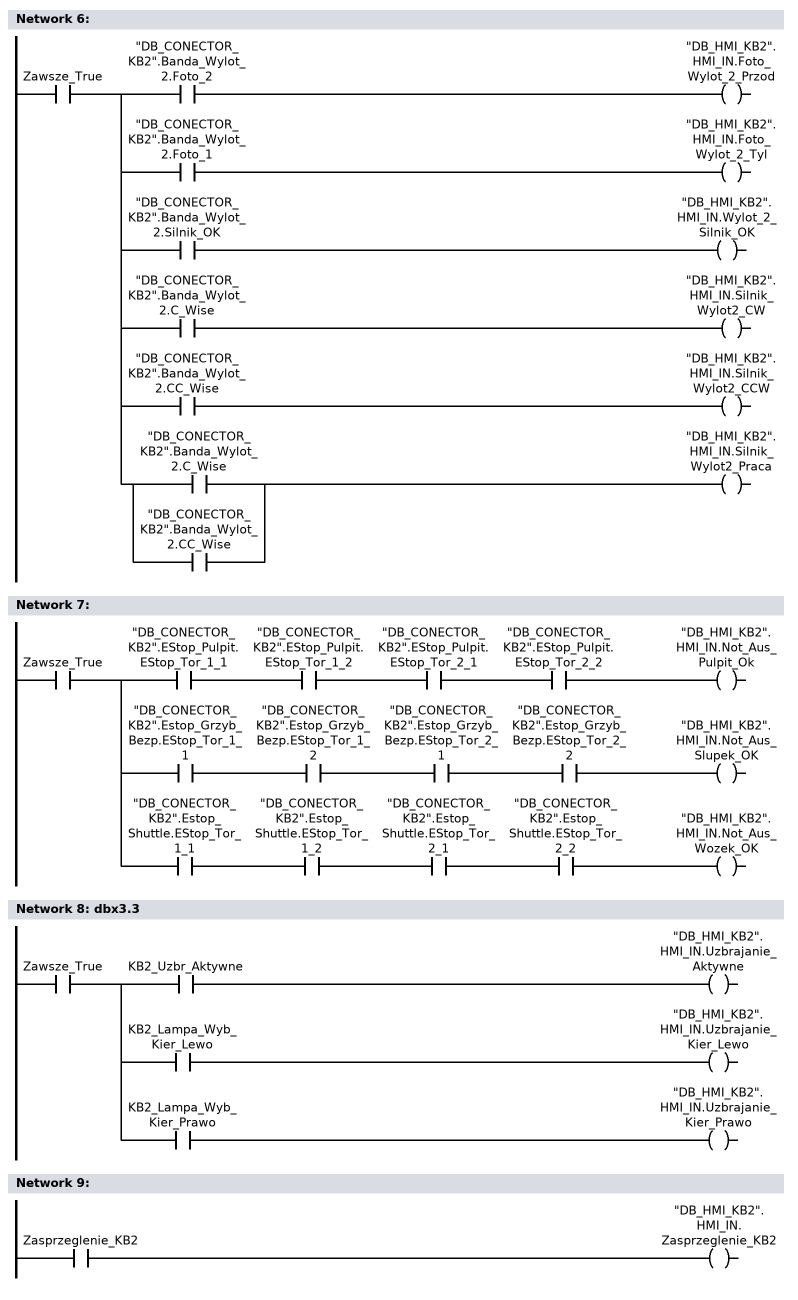
[picture p297: FC_HMI_KB2 networks 6-9]
NETWORK
TITLE =
//wylot 2
      A     "Zawsze_True";
      =     L 0.0;
      A     L 0.0;
      A     "DB_CONECTOR_KB2".Banda_Wylot_2.Foto_2;
      =     "DB_HMI_KB2".HMI_IN.Foto_Wylot_2_Przod;
      A     L 0.0;
      A     "DB_CONECTOR_KB2".Banda_Wylot_2.Foto_1;
      =     "DB_HMI_KB2".HMI_IN.Foto_Wylot_2_Tyl;
      A     L 0.0;
      A     "DB_CONECTOR_KB2".Banda_Wylot_2.Silnik_OK;
      =     "DB_HMI_KB2".HMI_IN.Wylot_2_Silnik_OK;
      A     L 0.0;
      A     "DB_CONECTOR_KB2".Banda_Wylot_2.C_Wise;
      =     "DB_HMI_KB2".HMI_IN.Silnik_Wylot2_CW;
      A     L 0.0;
      A     "DB_CONECTOR_KB2".Banda_Wylot_2.CC_Wise;
      =     "DB_HMI_KB2".HMI_IN.Silnik_Wylot2_CCW;
      A     L 0.0;
      A(;
      O     "DB_CONECTOR_KB2".Banda_Wylot_2.C_Wise;
      O     "DB_CONECTOR_KB2".Banda_Wylot_2.CC_Wise;
      );
      =     "DB_HMI_KB2".HMI_IN.Silnik_Wylot2_Praca;
NETWORK
TITLE =
//Not Aus pulpit
//
      A     "Zawsze_True";
      =     L 0.0;
      A     L 0.0;
      A     "DB_CONECTOR_KB2".EStop_Pulpit.EStop_Tor_1_1;
      A     "DB_CONECTOR_KB2".EStop_Pulpit.EStop_Tor_1_2;
      A     "DB_CONECTOR_KB2".EStop_Pulpit.EStop_Tor_2_1;
      A     "DB_CONECTOR_KB2".EStop_Pulpit.EStop_Tor_2_2;
      =     "DB_HMI_KB2".HMI_IN.Not_Aus_Pulpit_Ok;
      A     L 0.0;
      A     "DB_CONECTOR_KB2".Estop_Grzyb_Bezp.EStop_Tor_1_1;
      A     "DB_CONECTOR_KB2".Estop_Grzyb_Bezp.EStop_Tor_1_2;
      A     "DB_CONECTOR_KB2".Estop_Grzyb_Bezp.EStop_Tor_2_1;
      A     "DB_CONECTOR_KB2".Estop_Grzyb_Bezp.EStop_Tor_2_2;
      =     "DB_HMI_KB2".HMI_IN.Not_Aus_Slupek_OK;
      A     L 0.0;
      A     "DB_CONECTOR_KB2".Estop_Shuttle.EStop_Tor_1_1;
      A     "DB_CONECTOR_KB2".Estop_Shuttle.EStop_Tor_1_2;
      A     "DB_CONECTOR_KB2".Estop_Shuttle.EStop_Tor_2_1;
      A     "DB_CONECTOR_KB2".Estop_Shuttle.EStop_Tor_2_2;
      =     "DB_HMI_KB2".HMI_IN.Not_Aus_Wozek_OK;
NETWORK
TITLE = dbx3.3
//Uzbrajanie Aktywne
      A     "Zawsze_True";
      =     L 0.0;
      A     L 0.0;
      A     "KB2_Uzbr_Aktywne";
      =     "DB_HMI_KB2".HMI_IN.Uzbrajanie_Aktywne;
      A     L 0.0;
      A     "KB2_Lampa_Wyb_Kier_Lewo";
      =     "DB_HMI_KB2".HMI_IN.Uzbrajanie_Kier_Lewo;
      A     L 0.0;
      A     "KB2_Lampa_Wyb_Kier_Prawo";
      =     "DB_HMI_KB2".HMI_IN.Uzbrajanie_Kier_Prawo;
NETWORK
TITLE =
//Marka Zasprzeglenia KB2
      A     "Zasprzeglenie_KB2";
      =     "DB_HMI_KB2".HMI_IN.Zasprzeglenie_KB2;
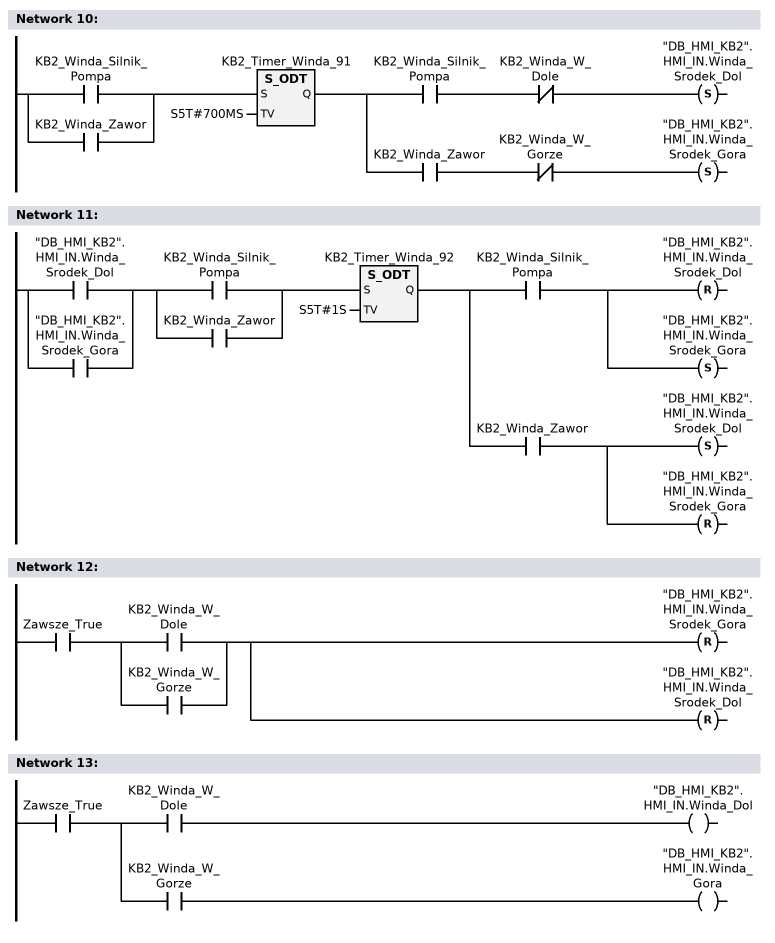
NETWORK
TITLE =
//Animacja windy
      A(;
      O     "KB2_Winda_Silnik_Pompa";
      O     "KB2_Winda_Zawor";
      );
      L     S5T#700MS;
      SD    "KB2_Timer_Winda_91";
      NOP   0;
      NOP   0;
      NOP   0;
      A     "KB2_Timer_Winda_91";
      =     L 0.0;
      A     L 0.0;
      A     "KB2_Winda_Silnik_Pompa";
      AN    "KB2_Winda_W_Dole";
      S     "DB_HMI_KB2".HMI_IN.Winda_Srodek_Dol;
      A     L 0.0;
      A     "KB2_Winda_Zawor";
      AN    "KB2_Winda_W_Gorze";
      S     "DB_HMI_KB2".HMI_IN.Winda_Srodek_Gora;
NETWORK
TITLE =
      A(;
      O     "DB_HMI_KB2".HMI_IN.Winda_Srodek_Dol;
      O     "DB_HMI_KB2".HMI_IN.Winda_Srodek_Gora;
      );
      A(;
      O     "KB2_Winda_Silnik_Pompa";
      O     "KB2_Winda_Zawor";
      );
      L     S5T#1S;
      SD    "KB2_Timer_Winda_92";
      NOP   0;
      NOP   0;
      NOP   0;
      A     "KB2_Timer_Winda_92";
      =     L 0.0;
      A     L 0.0;
      A     "KB2_Winda_Silnik_Pompa";
      R     "DB_HMI_KB2".HMI_IN.Winda_Srodek_Dol;
      S     "DB_HMI_KB2".HMI_IN.Winda_Srodek_Gora;
      A     L 0.0;
      A     "KB2_Winda_Zawor";
      S     "DB_HMI_KB2".HMI_IN.Winda_Srodek_Dol;
      R     "DB_HMI_KB2".HMI_IN.Winda_Srodek_Gora;
NETWORK
TITLE =
//Kasowanie skrajne winda
      A     "Zawsze_True";
      A(;
      O     "KB2_Winda_W_Dole";
      O     "KB2_Winda_W_Gorze";
      );
      R     "DB_HMI_KB2".HMI_IN.Winda_Srodek_Gora;
      R     "DB_HMI_KB2".HMI_IN.Winda_Srodek_Dol;
NETWORK
TITLE =
      A     "Zawsze_True";
      =     L 0.0;
      A     L 0.0;
      A     "KB2_Winda_W_Dole";
      =     "DB_HMI_KB2".HMI_IN.Winda_Dol;
      A     L 0.0;
      A     "KB2_Winda_W_Gorze";
      =     "DB_HMI_KB2".HMI_IN.Winda_Gora;
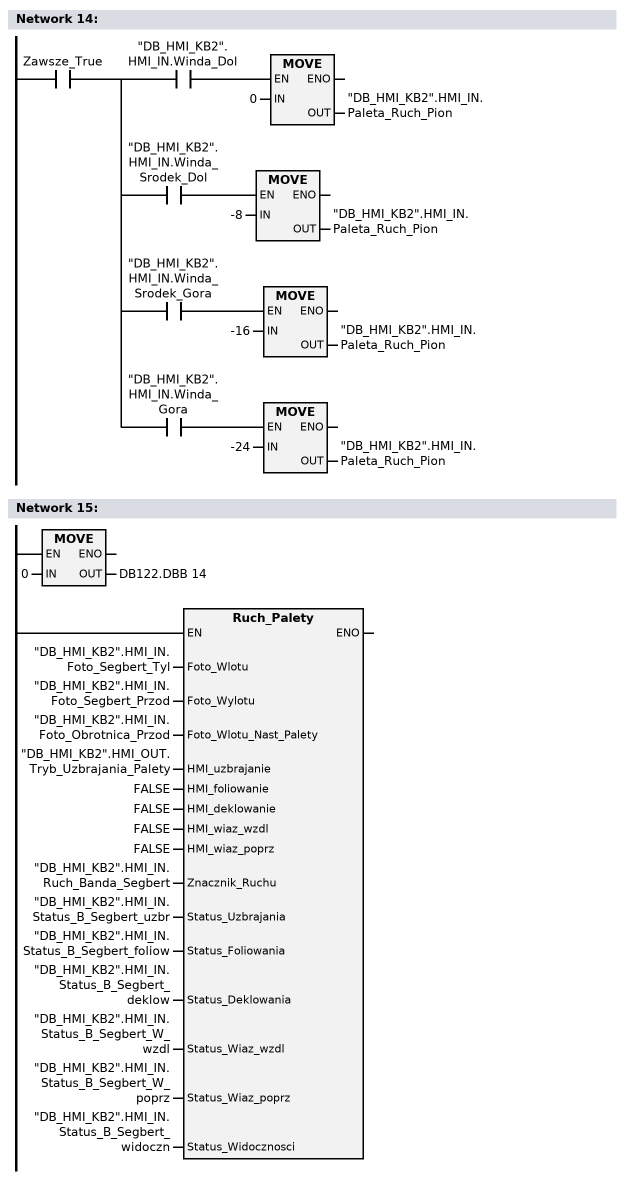
NETWORK
TITLE =
      A     "Zawsze_True";
      =     L 0.0;
      A     L 0.0;
      A     "DB_HMI_KB2".HMI_IN.Winda_Dol;
      JNB   _001;
      L     0;
      T     "DB_HMI_KB2".HMI_IN.Paleta_Ruch_Pion;
_001: NOP   0;
      A     L 0.0;
      A     "DB_HMI_KB2".HMI_IN.Winda_Srodek_Dol;
      JNB   _002;
      L     -8;
      T     "DB_HMI_KB2".HMI_IN.Paleta_Ruch_Pion;
_002: NOP   0;
      A     L 0.0;
      A     "DB_HMI_KB2".HMI_IN.Winda_Srodek_Gora;
      JNB   _003;
      L     -16;
      T     "DB_HMI_KB2".HMI_IN.Paleta_Ruch_Pion;
_003: NOP   0;
      A     L 0.0;
      A     "DB_HMI_KB2".HMI_IN.Winda_Gora;
      JNB   _004;
      L     -24;
      T     "DB_HMI_KB2".HMI_IN.Paleta_Ruch_Pion;
_004: NOP   0;
NETWORK
TITLE =
////Banda Segbert
      L     0;
      T     DB122.DBB 14;
      CALL  "Ruch_Palety" (
           Foto_Wlotu               := "DB_HMI_KB2".HMI_IN.Foto_Segbert_Tyl,
           Foto_Wylotu              := "DB_HMI_KB2".HMI_IN.Foto_Segbert_Przod,
           Foto_Wlotu_Nast_Palety   := "DB_HMI_KB2".HMI_IN.Foto_Obrotnica_Przod,
           HMI_uzbrajanie           := "DB_HMI_KB2".HMI_OUT.Tryb_Uzbrajania_Palety,
           HMI_foliowanie           := FALSE,
           HMI_deklowanie           := FALSE,
           HMI_wiaz_wzdl            := FALSE,
           HMI_wiaz_poprz           := FALSE,
           Znacznik_Ruchu           := "DB_HMI_KB2".HMI_IN.Ruch_Banda_Segbert,
           Status_Uzbrajania        := "DB_HMI_KB2".HMI_IN.Status_B_Segbert_uzbr,
           Status_Foliowania        := "DB_HMI_KB2".HMI_IN.Status_B_Segbert_foliow,
           Status_Deklowania        := "DB_HMI_KB2".HMI_IN.Status_B_Segbert_deklow,
           Status_Wiaz_wzdl         := "DB_HMI_KB2".HMI_IN.Status_B_Segbert_W_wzdl,
           Status_Wiaz_poprz        := "DB_HMI_KB2".HMI_IN.Status_B_Segbert_W_poprz,
           Status_Widocznosci       := "DB_HMI_KB2".HMI_IN.Status_B_Segbert_widoczn);
NETWORK
TITLE =
////Banda Obrotnica 0st
      L     0;
      T     DB122.DBB 15;
      A     DB122.DBX 7.0;
      JCN   et0;
      CALL  "Ruch_Palety" (
           Foto_Wlotu               := "DB_HMI_KB2".HMI_IN.Foto_Obrotnica_Przod,
           Foto_Wylotu              := "DB_HMI_KB2".HMI_IN.Foto_Obrotnica_Tyl,
           Foto_Wlotu_Nast_Palety   := "DB_HMI_KB2".HMI_IN.Foto_Winda_Tyl,
           HMI_uzbrajanie           := "DB_HMI_KB2".HMI_OUT.Tryb_Uzbrajania_Palety,
           HMI_foliowanie           := FALSE,
           HMI_deklowanie           := FALSE,
           HMI_wiaz_wzdl            := FALSE,
           HMI_wiaz_poprz           := FALSE,
           Znacznik_Ruchu           := "DB_HMI_KB2".HMI_IN.Ruch_Banda_Obrotnicy,
           Status_Uzbrajania        := "DB_HMI_KB2".HMI_IN.Status_B_Obr_0st_uzbr,
           Status_Foliowania        := "DB_HMI_KB2".HMI_IN.Status_B_Obr_0st_foliow,
           Status_Deklowania        := "DB_HMI_KB2".HMI_IN.Status_B_Obr_0st_deklow,
           Status_Wiaz_wzdl         := "DB_HMI_KB2".HMI_IN.Status_B_Obr_0st_W_wzdl,
           Status_Wiaz_poprz        := "DB_HMI_KB2".HMI_IN.Status_B_Obr_0st_W_poprz,
           Status_Widocznosci       := "DB_HMI_KB2".HMI_IN.Status_B_Obr_0st_widoczn);
      JU    ok0;
et0:  SET;
      R     "DB_HMI_KB2".HMI_IN.Status_B_Obr_0st_widoczn;
ok0:  NOP   0;
NETWORK
TITLE =
////Banda Obrotnica 90st
      L     0;
      T     DB122.DBB 19;
      A     DB122.DBX 8.0;
      JCN   et90;
      CALL  "Ruch_Palety" (
           Foto_Wlotu               := "DB_HMI_KB2".HMI_IN.Foto_Obrotnica_Przod,
           Foto_Wylotu              := "DB_HMI_KB2".HMI_IN.Foto_Obrotnica_Tyl,
           Foto_Wlotu_Nast_Palety   := "DB_HMI_KB2".HMI_IN.Foto_Wylot_2_Tyl,
           HMI_uzbrajanie           := "DB_HMI_KB2".HMI_OUT.Tryb_Uzbrajania_Palety,
           HMI_foliowanie           := FALSE,
           HMI_deklowanie           := FALSE,
           HMI_wiaz_wzdl            := FALSE,
           HMI_wiaz_poprz           := FALSE,
           Znacznik_Ruchu           := "DB_HMI_KB2".HMI_IN.Ruch_Banda_Obrotnicy,
           Status_Uzbrajania        := "DB_HMI_KB2".HMI_IN.Status_B_Obr_90st_uzbr,
           Status_Foliowania        := "DB_HMI_KB2".HMI_IN.Status_B_Obr_90st_foliow,
           Status_Deklowania        := "DB_HMI_KB2".HMI_IN.Status_B_Obr_90st_deklow,
           Status_Wiaz_wzdl         := "DB_HMI_KB2".HMI_IN.Status_B_Obr_90st_W_wzdl,
           Status_Wiaz_poprz        := "DB_HMI_KB2".HMI_IN.Status_B_Obr_90st_W_popr,
           Status_Widocznosci       := "DB_HMI_KB2".HMI_IN.Status_B_Obr_90st_widocz);
      JU    ok90;
et90: SET;
      R     "DB_HMI_KB2".HMI_IN.Status_B_Obr_90st_widocz;
ok90: NOP   0;
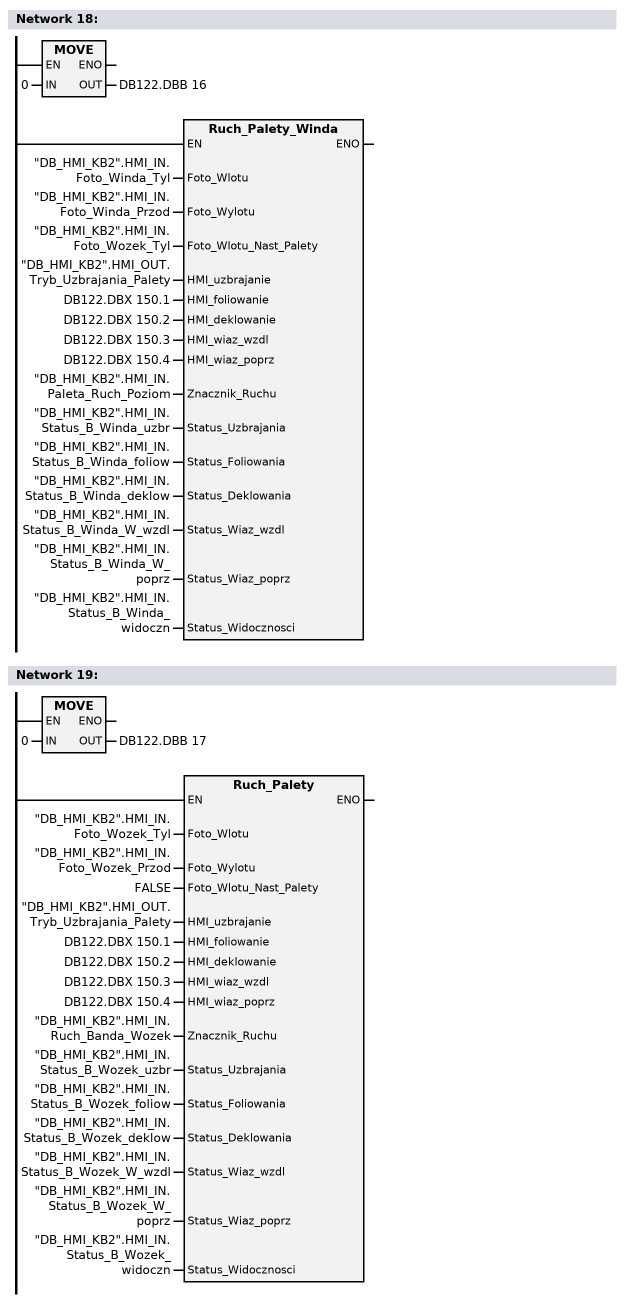
NETWORK
TITLE =
////Banda Winda
      L     0;
      T     DB122.DBB 16;
      CALL  "Ruch_Palety_Winda" (
           Foto_Wlotu               := "DB_HMI_KB2".HMI_IN.Foto_Winda_Tyl,
           Foto_Wylotu              := "DB_HMI_KB2".HMI_IN.Foto_Winda_Przod,
           Foto_Wlotu_Nast_Palety   := "DB_HMI_KB2".HMI_IN.Foto_Wozek_Tyl,
           HMI_uzbrajanie           := "DB_HMI_KB2".HMI_OUT.Tryb_Uzbrajania_Palety,
           HMI_foliowanie           := DB122.DBX 150.1,
           HMI_deklowanie           := DB122.DBX 150.2,
           HMI_wiaz_wzdl            := DB122.DBX 150.3,
           HMI_wiaz_poprz           := DB122.DBX 150.4,
           Znacznik_Ruchu           := "DB_HMI_KB2".HMI_IN.Paleta_Ruch_Poziom,
           Status_Uzbrajania        := "DB_HMI_KB2".HMI_IN.Status_B_Winda_uzbr,
           Status_Foliowania        := "DB_HMI_KB2".HMI_IN.Status_B_Winda_foliow,
           Status_Deklowania        := "DB_HMI_KB2".HMI_IN.Status_B_Winda_deklow,
           Status_Wiaz_wzdl         := "DB_HMI_KB2".HMI_IN.Status_B_Winda_W_wzdl,
           Status_Wiaz_poprz        := "DB_HMI_KB2".HMI_IN.Status_B_Winda_W_poprz,
           Status_Widocznosci       := "DB_HMI_KB2".HMI_IN.Status_B_Winda_widoczn);
NETWORK
TITLE =
////Banda Wozek
      L     0;
      T     DB122.DBB 17;
      CALL  "Ruch_Palety" (
           Foto_Wlotu               := "DB_HMI_KB2".HMI_IN.Foto_Wozek_Tyl,
           Foto_Wylotu              := "DB_HMI_KB2".HMI_IN.Foto_Wozek_Przod,
           Foto_Wlotu_Nast_Palety   := FALSE,
           HMI_uzbrajanie           := "DB_HMI_KB2".HMI_OUT.Tryb_Uzbrajania_Palety,
           HMI_foliowanie           := DB122.DBX 150.1,
           HMI_deklowanie           := DB122.DBX 150.2,
           HMI_wiaz_wzdl            := DB122.DBX 150.3,
           HMI_wiaz_poprz           := DB122.DBX 150.4,
           Znacznik_Ruchu           := "DB_HMI_KB2".HMI_IN.Ruch_Banda_Wozek,
           Status_Uzbrajania        := "DB_HMI_KB2".HMI_IN.Status_B_Wozek_uzbr,
           Status_Foliowania        := "DB_HMI_KB2".HMI_IN.Status_B_Wozek_foliow,
           Status_Deklowania        := "DB_HMI_KB2".HMI_IN.Status_B_Wozek_deklow,
           Status_Wiaz_wzdl         := "DB_HMI_KB2".HMI_IN.Status_B_Wozek_W_wzdl,
           Status_Wiaz_poprz        := "DB_HMI_KB2".HMI_IN.Status_B_Wozek_W_poprz,
           Status_Widocznosci       := "DB_HMI_KB2".HMI_IN.Status_B_Wozek_widoczn);
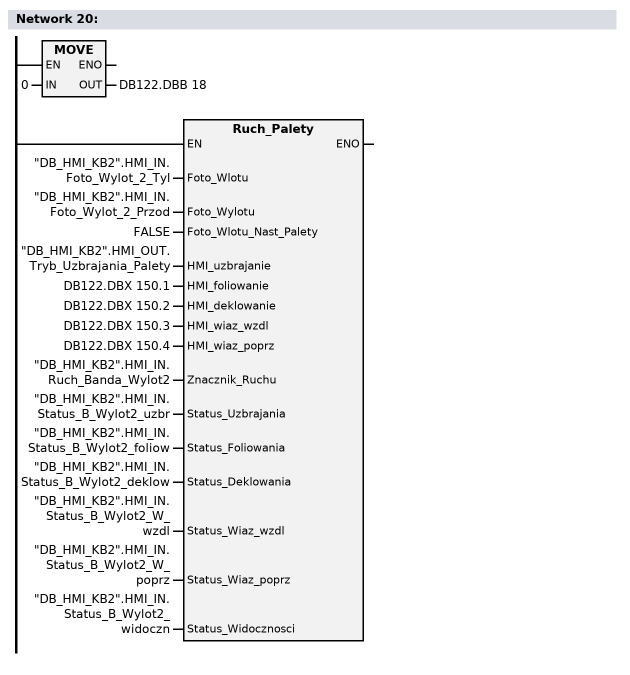
NETWORK
TITLE =
////Banda Wylot2
      L     0;
      T     DB122.DBB 18;
      CALL  "Ruch_Palety" (
           Foto_Wlotu               := "DB_HMI_KB2".HMI_IN.Foto_Wylot_2_Tyl,
           Foto_Wylotu              := "DB_HMI_KB2".HMI_IN.Foto_Wylot_2_Przod,
           Foto_Wlotu_Nast_Palety   := FALSE,
           HMI_uzbrajanie           := "DB_HMI_KB2".HMI_OUT.Tryb_Uzbrajania_Palety,
           HMI_foliowanie           := DB122.DBX 150.1,
           HMI_deklowanie           := DB122.DBX 150.2,
           HMI_wiaz_wzdl            := DB122.DBX 150.3,
           HMI_wiaz_poprz           := DB122.DBX 150.4,
           Znacznik_Ruchu           := "DB_HMI_KB2".HMI_IN.Ruch_Banda_Wylot2,
           Status_Uzbrajania        := "DB_HMI_KB2".HMI_IN.Status_B_Wylot2_uzbr,
           Status_Foliowania        := "DB_HMI_KB2".HMI_IN.Status_B_Wylot2_foliow,
           Status_Deklowania        := "DB_HMI_KB2".HMI_IN.Status_B_Wylot2_deklow,
           Status_Wiaz_wzdl         := "DB_HMI_KB2".HMI_IN.Status_B_Wylot2_W_wzdl,
           Status_Wiaz_poprz        := "DB_HMI_KB2".HMI_IN.Status_B_Wylot2_W_poprz,
           Status_Widocznosci       := "DB_HMI_KB2".HMI_IN.Status_B_Wylot2_widoczn);
END_FUNCTION

FUNCTION "FC_HMI_BUFF" : VOID	// FC 123
VERSION : 0.1
BEGIN
NETWORK
TITLE =
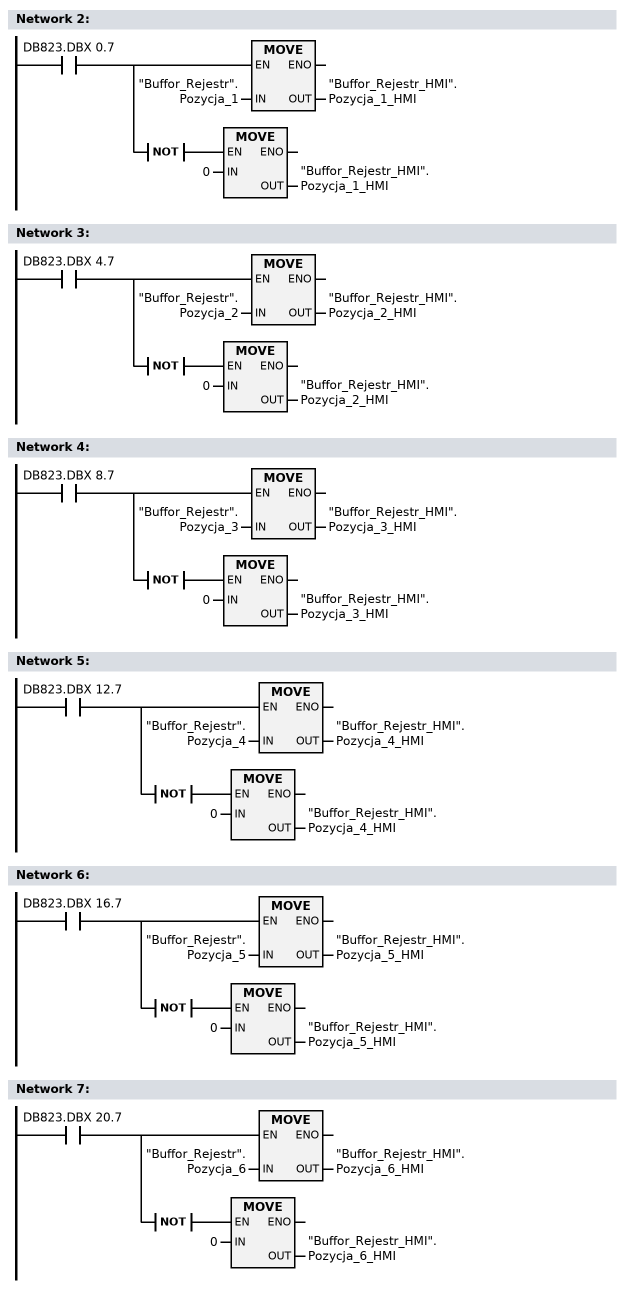
NETWORK
TITLE =
      A     DB823.DBX 0.7;
      =     L 0.0;
      A     L 0.0;
      JNB   _001;
      L     "Buffor_Rejestr".Pozycja_1;
      T     "Buffor_Rejestr_HMI".Pozycja_1_HMI;
_001: NOP   0;
      A     L 0.0;
      NOT;
      JNB   _008;
      L     0;
      T     "Buffor_Rejestr_HMI".Pozycja_1_HMI;
_008: NOP   0;
NETWORK
TITLE =
      A     DB823.DBX 4.7;
      =     L 0.0;
      A     L 0.0;
      JNB   _009;
      L     "Buffor_Rejestr".Pozycja_2;
      T     "Buffor_Rejestr_HMI".Pozycja_2_HMI;
_009: NOP   0;
      A     L 0.0;
      NOT;
      JNB   _00a;
      L     0;
      T     "Buffor_Rejestr_HMI".Pozycja_2_HMI;
_00a: NOP   0;
NETWORK
TITLE =
      A     DB823.DBX 8.7;
      =     L 0.0;
      A     L 0.0;
      JNB   _00b;
      L     "Buffor_Rejestr".Pozycja_3;
      T     "Buffor_Rejestr_HMI".Pozycja_3_HMI;
_00b: NOP   0;
      A     L 0.0;
      NOT;
      JNB   _00c;
      L     0;
      T     "Buffor_Rejestr_HMI".Pozycja_3_HMI;
_00c: NOP   0;
NETWORK
TITLE =
      A     DB823.DBX 12.7;
      =     L 0.0;
      A     L 0.0;
      JNB   _00d;
      L     "Buffor_Rejestr".Pozycja_4;
      T     "Buffor_Rejestr_HMI".Pozycja_4_HMI;
_00d: NOP   0;
      A     L 0.0;
      NOT;
      JNB   _00e;
      L     0;
      T     "Buffor_Rejestr_HMI".Pozycja_4_HMI;
_00e: NOP   0;
NETWORK
TITLE =
      A     DB823.DBX 16.7;
      =     L 0.0;
      A     L 0.0;
      JNB   _00f;
      L     "Buffor_Rejestr".Pozycja_5;
      T     "Buffor_Rejestr_HMI".Pozycja_5_HMI;
_00f: NOP   0;
      A     L 0.0;
      NOT;
      JNB   _010;
      L     0;
      T     "Buffor_Rejestr_HMI".Pozycja_5_HMI;
_010: NOP   0;
NETWORK
TITLE =
      A     DB823.DBX 20.7;
      =     L 0.0;
      A     L 0.0;
      JNB   _011;
      L     "Buffor_Rejestr".Pozycja_6;
      T     "Buffor_Rejestr_HMI".Pozycja_6_HMI;
_011: NOP   0;
      A     L 0.0;
      NOT;
      JNB   _012;
      L     0;
      T     "Buffor_Rejestr_HMI".Pozycja_6_HMI;
_012: NOP   0;
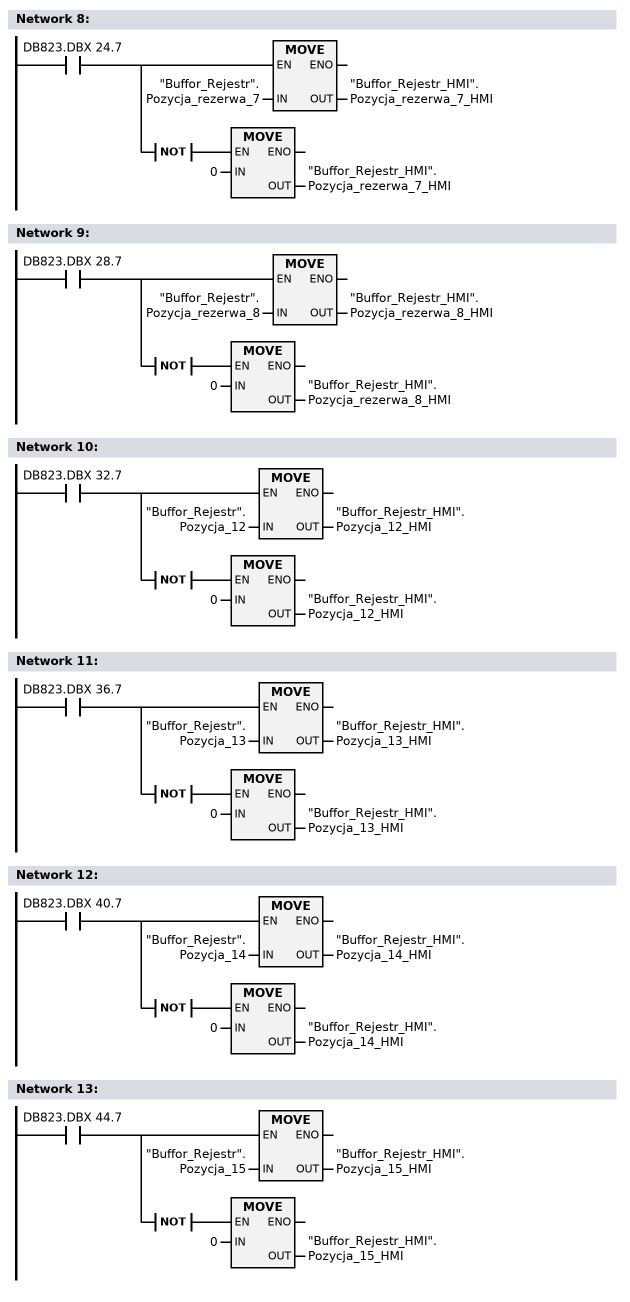
NETWORK
TITLE =
      A     DB823.DBX 24.7;
      =     L 0.0;
      A     L 0.0;
      JNB   _013;
      L     "Buffor_Rejestr".Pozycja_rezerwa_7;
      T     "Buffor_Rejestr_HMI".Pozycja_rezerwa_7_HMI;
_013: NOP   0;
      A     L 0.0;
      NOT;
      JNB   _014;
      L     0;
      T     "Buffor_Rejestr_HMI".Pozycja_rezerwa_7_HMI;
_014: NOP   0;
NETWORK
TITLE =
      A     DB823.DBX 28.7;
      =     L 0.0;
      A     L 0.0;
      JNB   _015;
      L     "Buffor_Rejestr".Pozycja_rezerwa_8;
      T     "Buffor_Rejestr_HMI".Pozycja_rezerwa_8_HMI;
_015: NOP   0;
      A     L 0.0;
      NOT;
      JNB   _016;
      L     0;
      T     "Buffor_Rejestr_HMI".Pozycja_rezerwa_8_HMI;
_016: NOP   0;
NETWORK
TITLE =
      A     DB823.DBX 32.7;
      =     L 0.0;
      A     L 0.0;
      JNB   _017;
      L     "Buffor_Rejestr".Pozycja_12;
      T     "Buffor_Rejestr_HMI".Pozycja_12_HMI;
_017: NOP   0;
      A     L 0.0;
      NOT;
      JNB   _018;
      L     0;
      T     "Buffor_Rejestr_HMI".Pozycja_12_HMI;
_018: NOP   0;
NETWORK
TITLE =
      A     DB823.DBX 36.7;
      =     L 0.0;
      A     L 0.0;
      JNB   _019;
      L     "Buffor_Rejestr".Pozycja_13;
      T     "Buffor_Rejestr_HMI".Pozycja_13_HMI;
_019: NOP   0;
      A     L 0.0;
      NOT;
      JNB   _01a;
      L     0;
      T     "Buffor_Rejestr_HMI".Pozycja_13_HMI;
_01a: NOP   0;
NETWORK
TITLE =
      A     DB823.DBX 40.7;
      =     L 0.0;
      A     L 0.0;
      JNB   _01b;
      L     "Buffor_Rejestr".Pozycja_14;
      T     "Buffor_Rejestr_HMI".Pozycja_14_HMI;
_01b: NOP   0;
      A     L 0.0;
      NOT;
      JNB   _01c;
      L     0;
      T     "Buffor_Rejestr_HMI".Pozycja_14_HMI;
_01c: NOP   0;
NETWORK
TITLE =
      A     DB823.DBX 44.7;
      =     L 0.0;
      A     L 0.0;
      JNB   _01d;
      L     "Buffor_Rejestr".Pozycja_15;
      T     "Buffor_Rejestr_HMI".Pozycja_15_HMI;
_01d: NOP   0;
      A     L 0.0;
      NOT;
      JNB   _01e;
      L     0;
      T     "Buffor_Rejestr_HMI".Pozycja_15_HMI;
_01e: NOP   0;
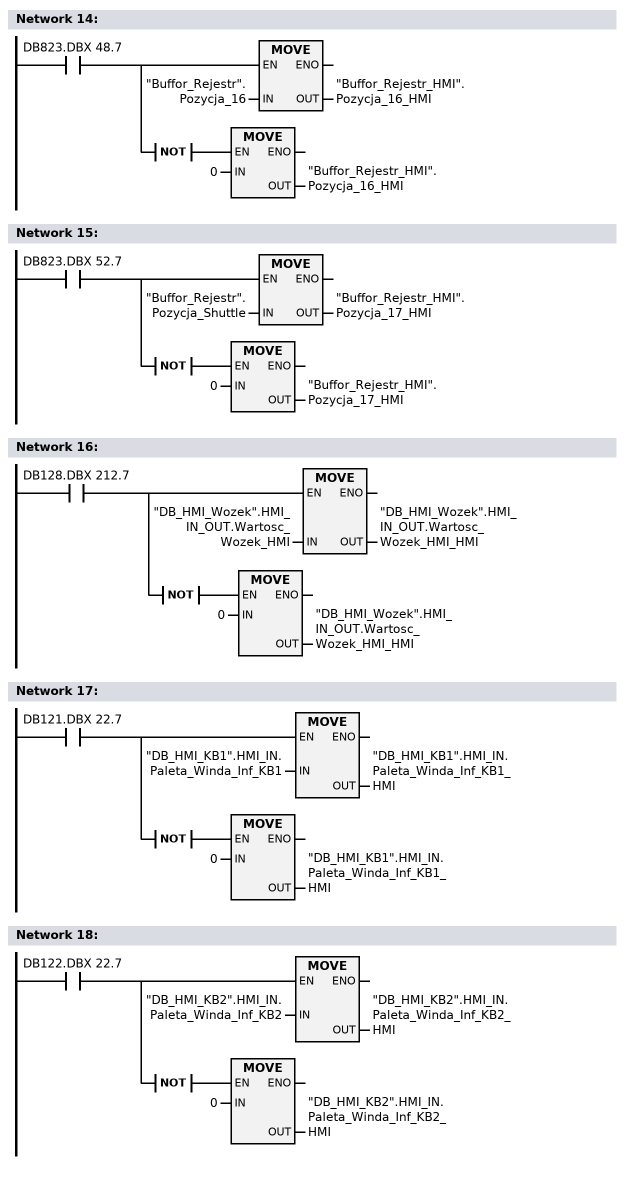
NETWORK
TITLE =
      A     DB823.DBX 48.7;
      =     L 0.0;
      A     L 0.0;
      JNB   _01f;
      L     "Buffor_Rejestr".Pozycja_16;
      T     "Buffor_Rejestr_HMI".Pozycja_16_HMI;
_01f: NOP   0;
      A     L 0.0;
      NOT;
      JNB   _020;
      L     0;
      T     "Buffor_Rejestr_HMI".Pozycja_16_HMI;
_020: NOP   0;
NETWORK
TITLE =
      A     DB823.DBX 52.7;
      =     L 0.0;
      A     L 0.0;
      JNB   _021;
      L     "Buffor_Rejestr".Pozycja_Shuttle;
      T     "Buffor_Rejestr_HMI".Pozycja_17_HMI;
_021: NOP   0;
      A     L 0.0;
      NOT;
      JNB   _022;
      L     0;
      T     "Buffor_Rejestr_HMI".Pozycja_17_HMI;
_022: NOP   0;
NETWORK
TITLE =
      A     DB128.DBX 212.7;
      =     L 0.0;
      A     L 0.0;
      JNB   _023;
      L     "DB_HMI_Wozek".HMI_IN_OUT.Wartosc_Wozek_HMI;
      T     "DB_HMI_Wozek".HMI_IN_OUT.Wartosc_Wozek_HMI_HMI;
_023: NOP   0;
      A     L 0.0;
      NOT;
      JNB   _024;
      L     0;
      T     "DB_HMI_Wozek".HMI_IN_OUT.Wartosc_Wozek_HMI_HMI;
_024: NOP   0;
NETWORK
TITLE =
      A     DB121.DBX 22.7;
      =     L 0.0;
      A     L 0.0;
      JNB   _025;
      L     "DB_HMI_KB1".HMI_IN.Paleta_Winda_Inf_KB1;
      T     "DB_HMI_KB1".HMI_IN.Paleta_Winda_Inf_KB1_HMI;
_025: NOP   0;
      A     L 0.0;
      NOT;
      JNB   _026;
      L     0;
      T     "DB_HMI_KB1".HMI_IN.Paleta_Winda_Inf_KB1_HMI;
_026: NOP   0;
NETWORK
TITLE =
      A     DB122.DBX 22.7;
      =     L 0.0;
      A     L 0.0;
      JNB   _027;
      L     "DB_HMI_KB2".HMI_IN.Paleta_Winda_Inf_KB2;
      T     "DB_HMI_KB2".HMI_IN.Paleta_Winda_Inf_KB2_HMI;
_027: NOP   0;
      A     L 0.0;
      NOT;
      JNB   _028;
      L     0;
      T     "DB_HMI_KB2".HMI_IN.Paleta_Winda_Inf_KB2_HMI;
_028: NOP   0;
END_FUNCTION

FUNCTION "FC_HMI_WOZEK" : VOID	// FC 128
AUTHOR : Kng
NAME : Main
VERSION : 0.1
VAR_TEMP
  Temp_Help_1 : BOOL ;
END_VAR
BEGIN
NETWORK
TITLE =
//Ten Network celowo jest wolny
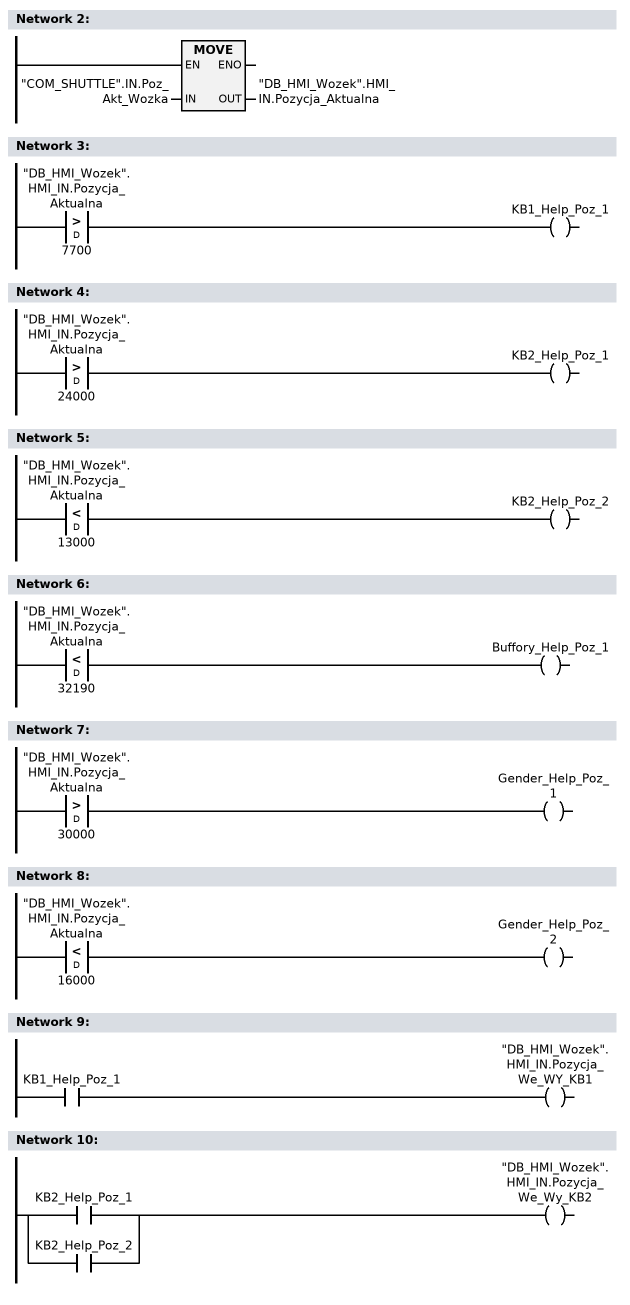
NETWORK
TITLE =
//Pozycja Aktualna
      L     "COM_SHUTTLE".IN.Poz_Akt_Wozka;
      T     "DB_HMI_Wozek".HMI_IN.Pozycja_Aktualna;
      NOP   0;
NETWORK
TITLE =
//wyznaczenie zakresu widzialnosci wozka na HMI dla KB1
      L     "DB_HMI_Wozek".HMI_IN.Pozycja_Aktualna;
      L     7700;
      >D;
      =     "KB1_Help_Poz_1";
NETWORK
TITLE =
//wyznaczenie zakresu widzialnosci wozka na HMI dla KB2
      L     "DB_HMI_Wozek".HMI_IN.Pozycja_Aktualna;
      L     24000;
      >D;
      =     "KB2_Help_Poz_1";
NETWORK
TITLE =
//wyznaczenie zakresu widzialnosci wozka na HMI dla KB2
      L     "DB_HMI_Wozek".HMI_IN.Pozycja_Aktualna;
      L     13000;
      <D;
      =     "KB2_Help_Poz_2";
NETWORK
TITLE =
//wyznaczenie zakresu widzialnosci wozka na HMI dla Buffory_Manual
//
      L     "DB_HMI_Wozek".HMI_IN.Pozycja_Aktualna;
      L     32190;
      <D;
      =     "Buffory_Help_Poz_1";
NETWORK
TITLE =
//wyznaczenie zakresu widzialnosci wozka na HMI dla Gender
      L     "DB_HMI_Wozek".HMI_IN.Pozycja_Aktualna;
      L     30000;
      >D;
      =     "Gender_Help_Poz_1";
NETWORK
TITLE =
//wyznaczenie zakresu widzialnosci wozka na HMI dla Gender
      L     "DB_HMI_Wozek".HMI_IN.Pozycja_Aktualna;
      L     16000;
      <D;
      =     "Gender_Help_Poz_2";
NETWORK
TITLE =
//wyznaczenie zakresu widzialnosci wozka na HMI dla KB1
      A     "KB1_Help_Poz_1";
      =     "DB_HMI_Wozek".HMI_IN.Pozycja_We_WY_KB1;
NETWORK
TITLE =
//wyznaczenie zakresu widzialnosci wozka na HMI dla KB2
      O     "KB2_Help_Poz_1";
      O     "KB2_Help_Poz_2";
      =     "DB_HMI_Wozek".HMI_IN.Pozycja_We_Wy_KB2;
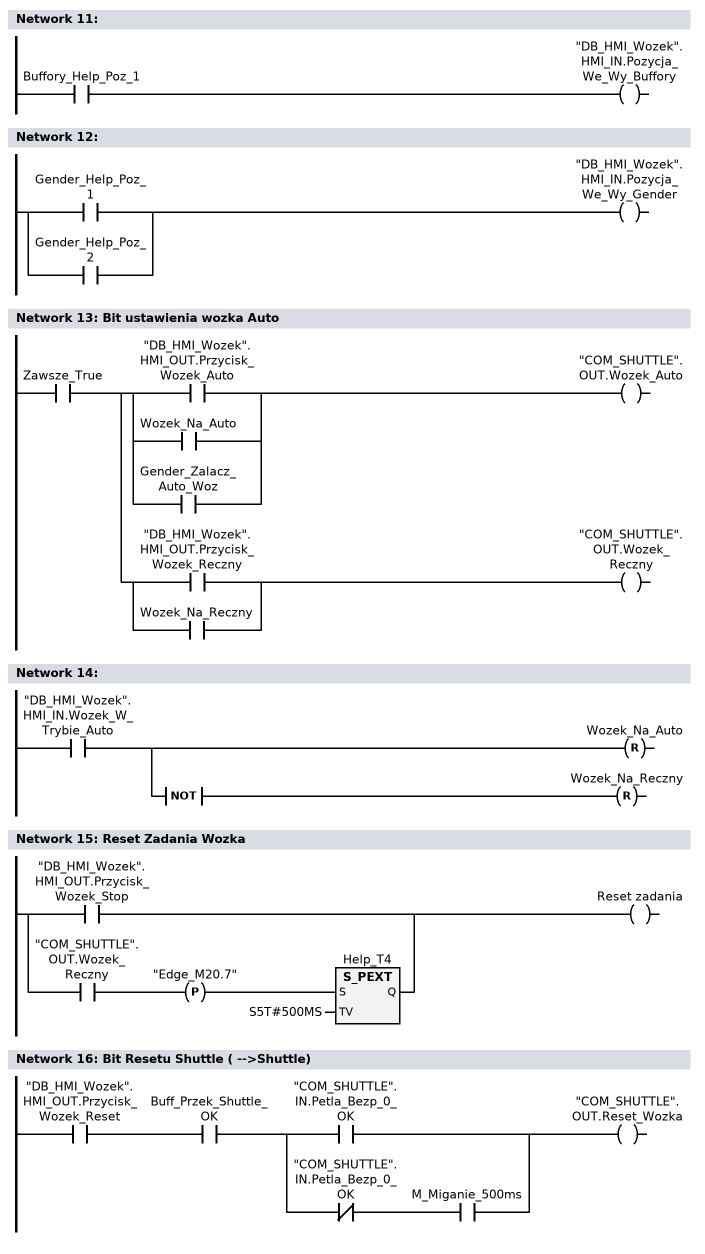
NETWORK
TITLE =
//wyznaczenie zakresu widzialnosci wozka na HMI dla Buffory_Manual
      A     "Buffory_Help_Poz_1";
      =     "DB_HMI_Wozek".HMI_IN.Pozycja_We_Wy_Buffory;
NETWORK
TITLE =
//wyznaczenie zakresu widzialnosci wozka na HMI dla Gender
      O     "Gender_Help_Poz_1";
      O     "Gender_Help_Poz_2";
      =     "DB_HMI_Wozek".HMI_IN.Pozycja_We_Wy_Gender;
NETWORK
TITLE = Bit ustawienia wozka Auto
//Wybranie trybu pracy wozka 
      A     "Zawsze_True";
      =     L 1.0;
      A     L 1.0;
      A(;
      O     "DB_HMI_Wozek".HMI_OUT.Przycisk_Wozek_Auto;
      O     "Wozek_Na_Auto";
      O     "Gender_Zalacz_Auto_Woz";
      );
      =     "COM_SHUTTLE".OUT.Wozek_Auto;
      A     L 1.0;
      A(;
      O     "DB_HMI_Wozek".HMI_OUT.Przycisk_Wozek_Reczny;
      O     "Wozek_Na_Reczny";
      );
      =     "COM_SHUTTLE".OUT.Wozek_Reczny;
NETWORK
TITLE =
//sprawdzenie w jakim trybie jest wozek
      A     "DB_HMI_Wozek".HMI_IN.Wozek_W_Trybie_Auto;
      =     L 1.0;
      A     L 1.0;
      BLD   102;
      R     "Wozek_Na_Auto";
      A     L 1.0;
      NOT;
      R     "Wozek_Na_Reczny";
NETWORK
TITLE = Reset Zadania Wozka
//Zatrzymanie zadania
//
      O     "DB_HMI_Wozek".HMI_OUT.Przycisk_Wozek_Stop;
      O(;
      A     "COM_SHUTTLE".OUT.Wozek_Reczny;
      FP    "Edge_M20.7";
      L     S5T#500MS;
      SE    "Help_T4";
      NOP   0;
      NOP   0;
      NOP   0;
      A     "Help_T4";
      );
      =     "Reset zadania";
NETWORK
TITLE = Bit Resetu Shuttle ( -->Shuttle)
//Reset bledow wozek
      A     "DB_HMI_Wozek".HMI_OUT.Przycisk_Wozek_Reset;
      A     "Buff_Przek_Shuttle_OK";
      A(;
      O     "COM_SHUTTLE".IN.Petla_Bezp_0_OK;
      O;
      AN    "COM_SHUTTLE".IN.Petla_Bezp_0_OK;
      A     "M_Miganie_500ms";
      );
      =     "COM_SHUTTLE".OUT.Reset_Wozka;
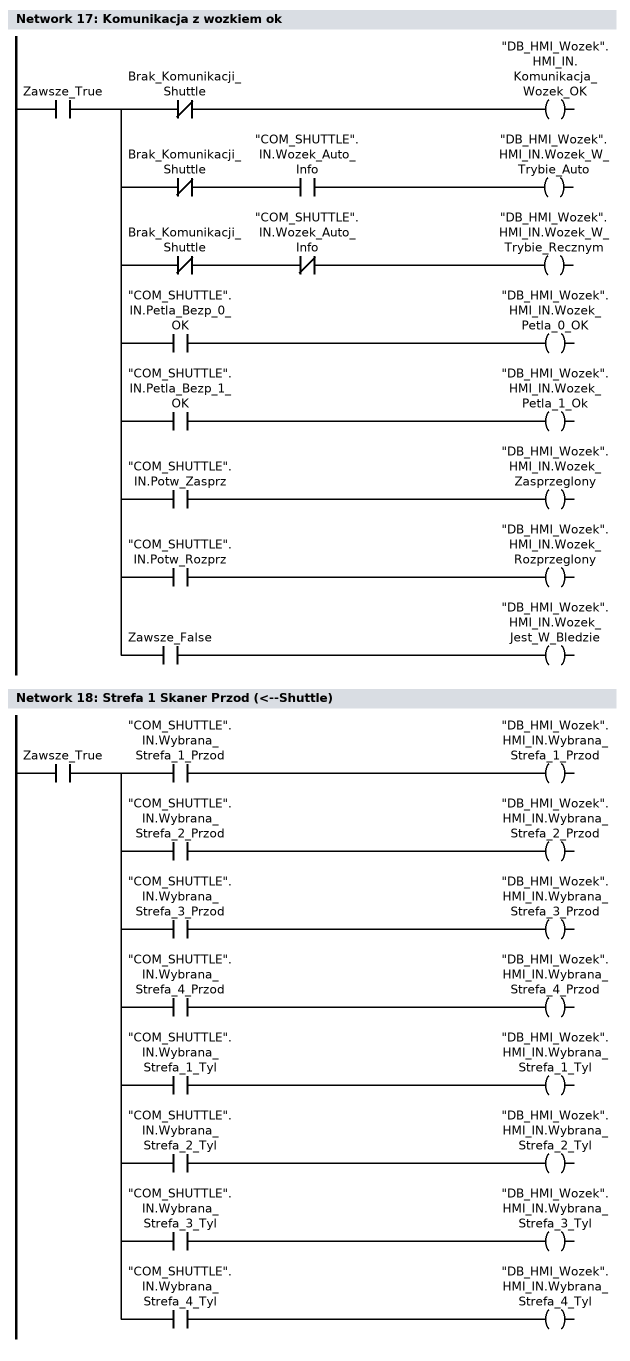
NETWORK
TITLE = Komunikacja z wozkiem ok 
//Potwierdzenie Trybu pracy wozek
      A     "Zawsze_True";
      =     L 1.0;
      A     L 1.0;
      AN    "Brak_Komunikacji_Shuttle";
      =     "DB_HMI_Wozek".HMI_IN.Komunikacja_Wozek_OK;
      A     L 1.0;
      AN    "Brak_Komunikacji_Shuttle";
      A     "COM_SHUTTLE".IN.Wozek_Auto_Info;
      =     "DB_HMI_Wozek".HMI_IN.Wozek_W_Trybie_Auto;
      A     L 1.0;
      AN    "Brak_Komunikacji_Shuttle";
      AN    "COM_SHUTTLE".IN.Wozek_Auto_Info;
      =     "DB_HMI_Wozek".HMI_IN.Wozek_W_Trybie_Recznym;
      A     L 1.0;
      A     "COM_SHUTTLE".IN.Petla_Bezp_0_OK;
      =     "DB_HMI_Wozek".HMI_IN.Wozek_Petla_0_OK;
      A     L 1.0;
      A     "COM_SHUTTLE".IN.Petla_Bezp_1_OK;
      =     "DB_HMI_Wozek".HMI_IN.Wozek_Petla_1_Ok;
      A     L 1.0;
      A     "COM_SHUTTLE".IN.Potw_Zasprz;
      =     "DB_HMI_Wozek".HMI_IN.Wozek_Zasprzeglony;
      A     L 1.0;
      A     "COM_SHUTTLE".IN.Potw_Rozprz;
      =     "DB_HMI_Wozek".HMI_IN.Wozek_Rozprzeglony;
      A     L 1.0;
      A     "Zawsze_False";
      =     "DB_HMI_Wozek".HMI_IN.Wozek_Jest_W_Bledzie;
NETWORK
TITLE = Strefa 1 Skaner Przod (<--Shuttle)
//Sprawdzenie ktora strefa jest aktywna
      A     "Zawsze_True";
      =     L 1.0;
      A     L 1.0;
      A     "COM_SHUTTLE".IN.Wybrana_Strefa_1_Przod;
      =     "DB_HMI_Wozek".HMI_IN.Wybrana_Strefa_1_Przod;
      A     L 1.0;
      A     "COM_SHUTTLE".IN.Wybrana_Strefa_2_Przod;
      =     "DB_HMI_Wozek".HMI_IN.Wybrana_Strefa_2_Przod;
      A     L 1.0;
      A     "COM_SHUTTLE".IN.Wybrana_Strefa_3_Przod;
      =     "DB_HMI_Wozek".HMI_IN.Wybrana_Strefa_3_Przod;
      A     L 1.0;
      A     "COM_SHUTTLE".IN.Wybrana_Strefa_4_Przod;
      =     "DB_HMI_Wozek".HMI_IN.Wybrana_Strefa_4_Przod;
      A     L 1.0;
      A     "COM_SHUTTLE".IN.Wybrana_Strefa_1_Tyl;
      =     "DB_HMI_Wozek".HMI_IN.Wybrana_Strefa_1_Tyl;
      A     L 1.0;
      A     "COM_SHUTTLE".IN.Wybrana_Strefa_2_Tyl;
      =     "DB_HMI_Wozek".HMI_IN.Wybrana_Strefa_2_Tyl;
      A     L 1.0;
      A     "COM_SHUTTLE".IN.Wybrana_Strefa_3_Tyl;
      =     "DB_HMI_Wozek".HMI_IN.Wybrana_Strefa_3_Tyl;
      A     L 1.0;
      A     "COM_SHUTTLE".IN.Wybrana_Strefa_4_Tyl;
      =     "DB_HMI_Wozek".HMI_IN.Wybrana_Strefa_4_Tyl;
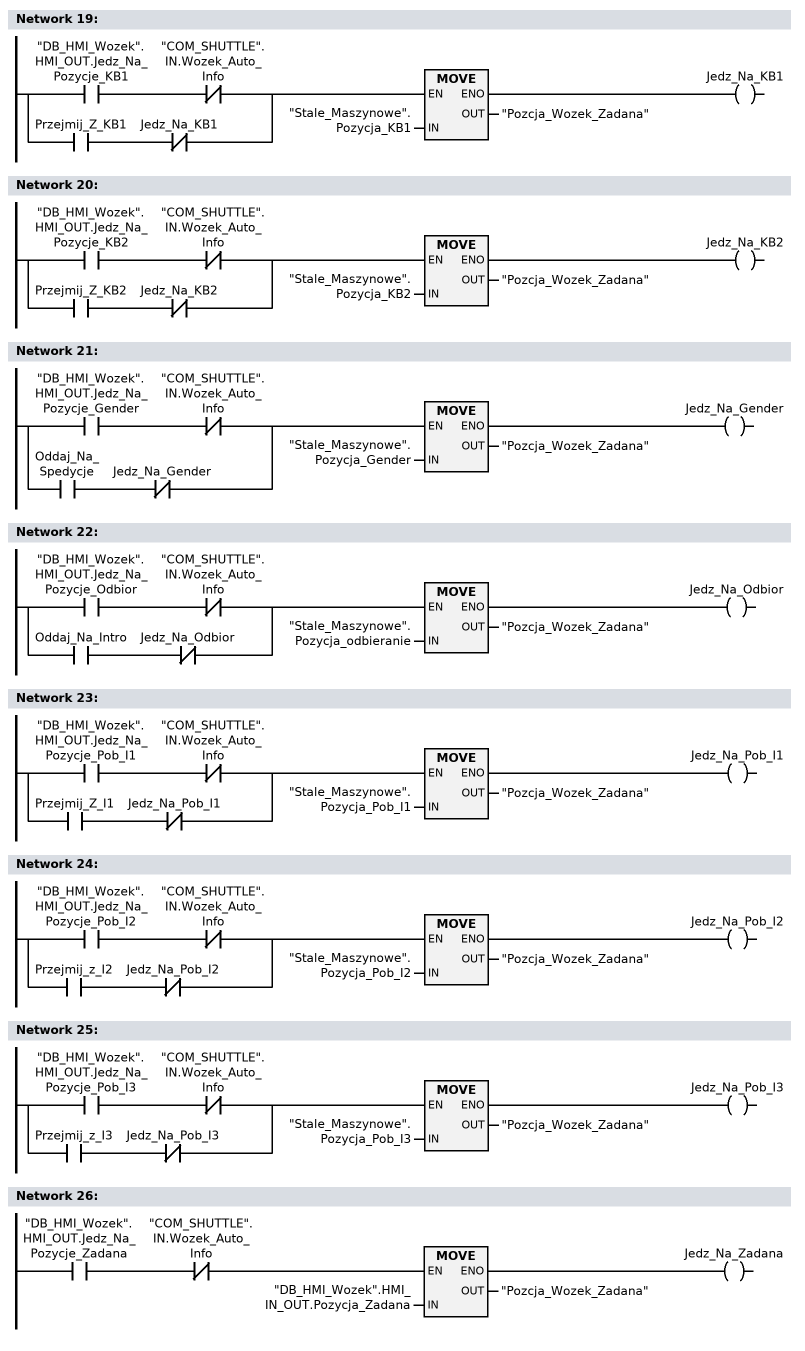
NETWORK
TITLE =
//Jedz na Kb1
//
      A(;
      A     "DB_HMI_Wozek".HMI_OUT.Jedz_Na_Pozycje_KB1;
      AN    "COM_SHUTTLE".IN.Wozek_Auto_Info;
      O;
      A     "Przejmij_Z_KB1";
      AN    "Jedz_Na_KB1";
      );
      JNB   _001;
      L     "Stale_Maszynowe".Pozycja_KB1;
      T     "Pozcja_Wozek_Zadana";
      SET;
      SAVE;
      CLR;
_001: A     BR;
      =     "Jedz_Na_KB1";
NETWORK
TITLE =
//Jedz na Kb2
//
//
      A(;
      A     "DB_HMI_Wozek".HMI_OUT.Jedz_Na_Pozycje_KB2;
      AN    "COM_SHUTTLE".IN.Wozek_Auto_Info;
      O;
      A     "Przejmij_Z_KB2";
      AN    "Jedz_Na_KB2";
      );
      JNB   _002;
      L     "Stale_Maszynowe".Pozycja_KB2;
      T     "Pozcja_Wozek_Zadana";
      SET;
      SAVE;
      CLR;
_002: A     BR;
      =     "Jedz_Na_KB2";
NETWORK
TITLE =
//Jedz na gender
//
//
      A(;
      A     "DB_HMI_Wozek".HMI_OUT.Jedz_Na_Pozycje_Gender;
      AN    "COM_SHUTTLE".IN.Wozek_Auto_Info;
      O;
      A     "Oddaj_Na_Spedycje";
      AN    "Jedz_Na_Gender";
      );
      JNB   _003;
      L     "Stale_Maszynowe".Pozycja_Gender;
      T     "Pozcja_Wozek_Zadana";
      SET;
      SAVE;
      CLR;
_003: A     BR;
      =     "Jedz_Na_Gender";
NETWORK
TITLE =
//Jedz na odbieranie
//
//
      A(;
      A     "DB_HMI_Wozek".HMI_OUT.Jedz_Na_Pozycje_Odbior;
      AN    "COM_SHUTTLE".IN.Wozek_Auto_Info;
      O;
      A     "Oddaj_Na_Intro";
      AN    "Jedz_Na_Odbior";
      );
      JNB   _004;
      L     "Stale_Maszynowe".Pozycja_odbieranie;
      T     "Pozcja_Wozek_Zadana";
      SET;
      SAVE;
      CLR;
_004: A     BR;
      =     "Jedz_Na_Odbior";
NETWORK
TITLE =
//Pobieranie I1
      A(;
      A     "DB_HMI_Wozek".HMI_OUT.Jedz_Na_Pozycje_Pob_I1;
      AN    "COM_SHUTTLE".IN.Wozek_Auto_Info;
      O;
      A     "Przejmij_Z_I1";
      AN    "Jedz_Na_Pob_I1";
      );
      JNB   _005;
      L     "Stale_Maszynowe".Pozycja_Pob_I1;
      T     "Pozcja_Wozek_Zadana";
      SET;
      SAVE;
      CLR;
_005: A     BR;
      =     "Jedz_Na_Pob_I1";
NETWORK
TITLE =
//Pobieranie I2
      A(;
      A     "DB_HMI_Wozek".HMI_OUT.Jedz_Na_Pozycje_Pob_I2;
      AN    "COM_SHUTTLE".IN.Wozek_Auto_Info;
      O;
      A     "Przejmij_z_I2";
      AN    "Jedz_Na_Pob_I2";
      );
      JNB   _006;
      L     "Stale_Maszynowe".Pozycja_Pob_I2;
      T     "Pozcja_Wozek_Zadana";
      SET;
      SAVE;
      CLR;
_006: A     BR;
      =     "Jedz_Na_Pob_I2";
NETWORK
TITLE =
//Pobieranie I3
      A(;
      A     "DB_HMI_Wozek".HMI_OUT.Jedz_Na_Pozycje_Pob_I3;
      AN    "COM_SHUTTLE".IN.Wozek_Auto_Info;
      O;
      A     "Przejmij_z_I3";
      AN    "Jedz_Na_Pob_I3";
      );
      JNB   _007;
      L     "Stale_Maszynowe".Pozycja_Pob_I3;
      T     "Pozcja_Wozek_Zadana";
      SET;
      SAVE;
      CLR;
_007: A     BR;
      =     "Jedz_Na_Pob_I3";
NETWORK
TITLE =
//Jedz na pozycje zadana z menu
      A     "DB_HMI_Wozek".HMI_OUT.Jedz_Na_Pozycje_Zadana;
      AN    "COM_SHUTTLE".IN.Wozek_Auto_Info;
      JNB   _008;
      L     "DB_HMI_Wozek".HMI_IN_OUT.Pozycja_Zadana;
      T     "Pozcja_Wozek_Zadana";
      SET;
      SAVE;
      CLR;
_008: A     BR;
      =     "Jedz_Na_Zadana";
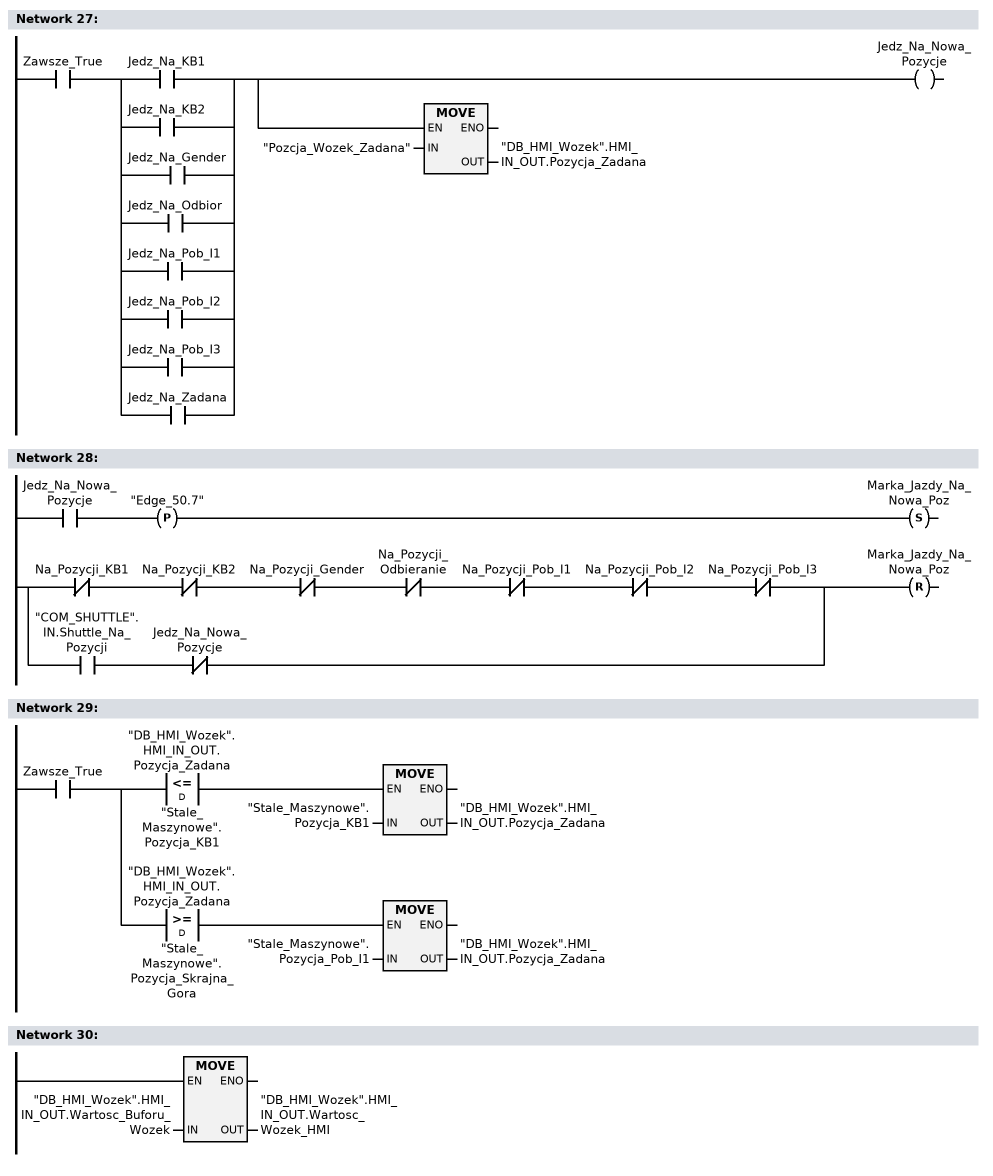
NETWORK
TITLE =
      A     "Zawsze_True";
      A(;
      O     "Jedz_Na_KB1";
      O     "Jedz_Na_KB2";
      O     "Jedz_Na_Gender";
      O     "Jedz_Na_Odbior";
      O     "Jedz_Na_Pob_I1";
      O     "Jedz_Na_Pob_I2";
      O     "Jedz_Na_Pob_I3";
      O     "Jedz_Na_Zadana";
      );
      =     L 1.0;
      A     L 1.0;
      BLD   102;
      =     "Jedz_Na_Nowa_Pozycje";
      A     L 1.0;
      JNB   _009;
      L     "Pozcja_Wozek_Zadana";
      T     "DB_HMI_Wozek".HMI_IN_OUT.Pozycja_Zadana;
_009: NOP   0;
NETWORK
TITLE =
//Funkcja lapania nowej pozycji
      A     "Jedz_Na_Nowa_Pozycje";
      FP    "Edge_50.7";
      S     "Marka_Jazdy_Na_Nowa_Poz";
      A(;
      AN    "Na_Pozycji_KB1";
      AN    "Na_Pozycji_KB2";
      AN    "Na_Pozycji_Gender";
      AN    "Na_Pozycji_Odbieranie";
      AN    "Na_Pozycji_Pob_I1";
      AN    "Na_Pozycji_Pob_I2";
      AN    "Na_Pozycji_Pob_I3";
      O;
      A     "COM_SHUTTLE".IN.Shuttle_Na_Pozycji;
      AN    "Jedz_Na_Nowa_Pozycje";
      );
      R     "Marka_Jazdy_Na_Nowa_Poz";
      NOP   0;
NETWORK
TITLE =
//Sprawdznie wartosci krytycznych
      A     "Zawsze_True";
      =     L 1.0;
      A     L 1.0;
      A(;
      L     "DB_HMI_Wozek".HMI_IN_OUT.Pozycja_Zadana;
      L     "Stale_Maszynowe".Pozycja_KB1;
      <=D;
      );
      JNB   _00a;
      L     "Stale_Maszynowe".Pozycja_KB1;
      T     "DB_HMI_Wozek".HMI_IN_OUT.Pozycja_Zadana;
_00a: NOP   0;
      A     L 1.0;
      A(;
      L     "DB_HMI_Wozek".HMI_IN_OUT.Pozycja_Zadana;
      L     "Stale_Maszynowe".Pozycja_Skrajna_Gora;
      >=D;
      );
      JNB   _00b;
      L     "Stale_Maszynowe".Pozycja_Pob_I1;
      T     "DB_HMI_Wozek".HMI_IN_OUT.Pozycja_Zadana;
_00b: NOP   0;
NETWORK
TITLE =
      L     "DB_HMI_Wozek".HMI_IN_OUT.Wartosc_Buforu_Wozek;
      T     "DB_HMI_Wozek".HMI_IN_OUT.Wartosc_Wozek_HMI;
      NOP   0;
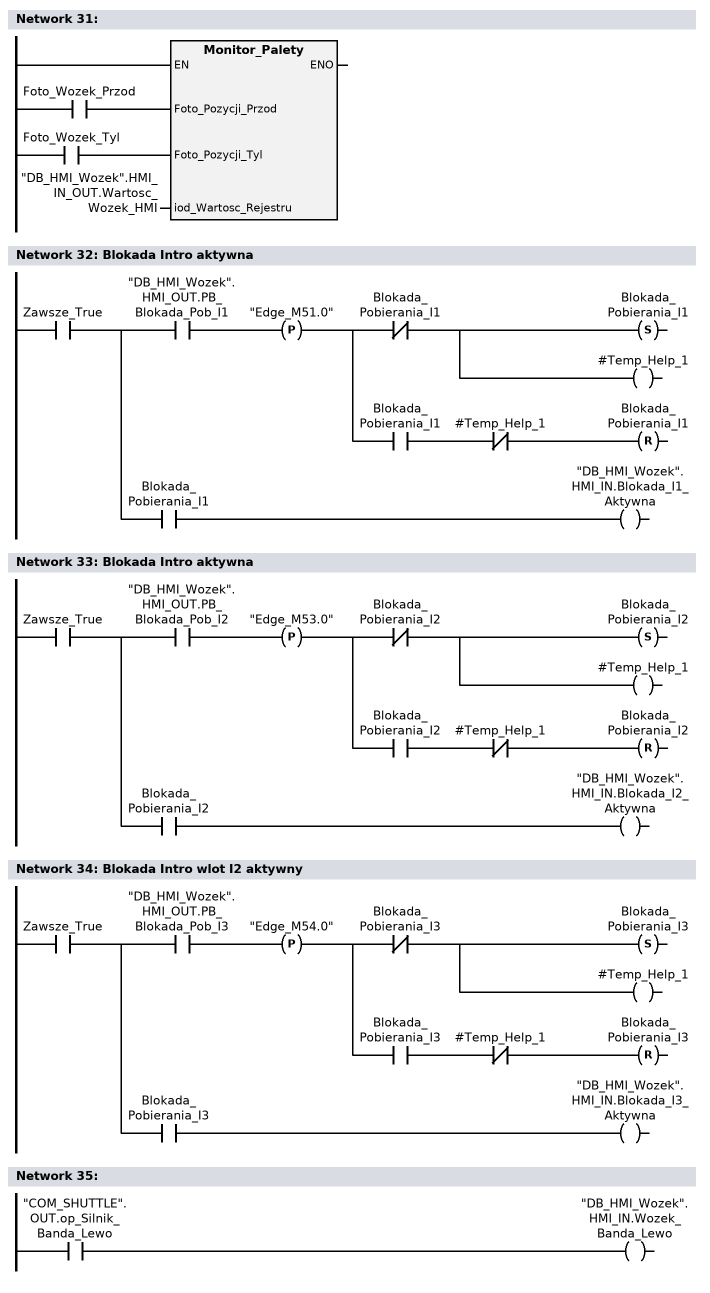
NETWORK
TITLE =
      A     "Foto_Wozek_Przod";
      =     L 1.0;
      BLD   103;
      A     "Foto_Wozek_Tyl";
      =     L 1.1;
      BLD   103;
      CALL  "Monitor_Palety" (
           Foto_Pozycji_Przod       := L 1.0,
           Foto_Pozycji_Tyl         := L 1.1,
           iod_Wartosc_Rejestru     := "DB_HMI_Wozek".HMI_IN_OUT.Wartosc_Wozek_HMI);
      NOP   0;
NETWORK
TITLE = Blokada Intro aktywna
//Blokada pobierania na intro
      A     "Zawsze_True";
      =     L 1.0;
      A     L 1.0;
      A     "DB_HMI_Wozek".HMI_OUT.PB_Blokada_Pob_I1;
      FP    "Edge_M51.0";
      =     L 1.1;
      A     L 1.1;
      AN    "Blokada_Pobierania_I1";
      S     "Blokada_Pobierania_I1";
      =     #Temp_Help_1;
      A     L 1.1;
      A     "Blokada_Pobierania_I1";
      AN    #Temp_Help_1;
      R     "Blokada_Pobierania_I1";
      A     L 1.0;
      A     "Blokada_Pobierania_I1";
      =     "DB_HMI_Wozek".HMI_IN.Blokada_I1_Aktywna;
NETWORK
TITLE = Blokada Intro aktywna
//Blokada pobierania na intro
      A     "Zawsze_True";
      =     L 1.0;
      A     L 1.0;
      A     "DB_HMI_Wozek".HMI_OUT.PB_Blokada_Pob_I2;
      FP    "Edge_M53.0";
      =     L 1.1;
      A     L 1.1;
      AN    "Blokada_Pobierania_I2";
      S     "Blokada_Pobierania_I2";
      =     #Temp_Help_1;
      A     L 1.1;
      A     "Blokada_Pobierania_I2";
      AN    #Temp_Help_1;
      R     "Blokada_Pobierania_I2";
      A     L 1.0;
      A     "Blokada_Pobierania_I2";
      =     "DB_HMI_Wozek".HMI_IN.Blokada_I2_Aktywna;
NETWORK
TITLE = Blokada Intro wlot I2 aktywny
      A     "Zawsze_True";
      =     L 1.0;
      A     L 1.0;
      A     "DB_HMI_Wozek".HMI_OUT.PB_Blokada_Pob_I3;
      FP    "Edge_M54.0";
      =     L 1.1;
      A     L 1.1;
      AN    "Blokada_Pobierania_I3";
      S     "Blokada_Pobierania_I3";
      =     #Temp_Help_1;
      A     L 1.1;
      A     "Blokada_Pobierania_I3";
      AN    #Temp_Help_1;
      R     "Blokada_Pobierania_I3";
      A     L 1.0;
      A     "Blokada_Pobierania_I3";
      =     "DB_HMI_Wozek".HMI_IN.Blokada_I3_Aktywna;
NETWORK
TITLE =
      A     "COM_SHUTTLE".OUT.op_Silnik_Banda_Lewo;
      =     "DB_HMI_Wozek".HMI_IN.Wozek_Banda_Lewo;
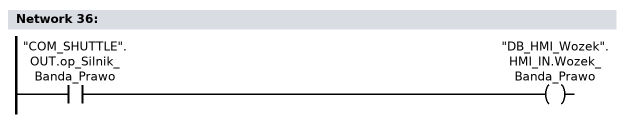
NETWORK
TITLE =
      A     "COM_SHUTTLE".OUT.op_Silnik_Banda_Prawo;
      =     "DB_HMI_Wozek".HMI_IN.Wozek_Banda_Prawo;
END_FUNCTION

FUNCTION "Funkcja_Zegara" : VOID	// FC 140
AUTHOR : Kng
NAME : HELP_FC
VERSION : 0.1
VAR_INPUT
  Timer_NR : TIMER ;
  Czas : S5TIME ;
END_VAR
VAR_IN_OUT
  Wyjscie : BOOL ;
END_VAR
BEGIN
NETWORK
TITLE =
      A     #Timer_NR;
      SAVE;
      NOT;
      L     #Czas;
      SD    #Timer_NR;
      X     BR;
      X     #Wyjscie;
      =     #Wyjscie;
END_FUNCTION

FUNCTION "Shuttle_Comand" : VOID	// FC 200
//Funkcja odpowiada za wymiane danych z wozkiem shuttle. Dane w formie struktury 
//sa zapisywane do bloku com. Blok jest strukturyzowany. Jego odwrotna wersja 
//znaduje sie w wozku.
AUTHOR : Kng
NAME : Fahren
VERSION : 0.1
BEGIN
NETWORK
TITLE =
//Ten Network celowo jest wolny
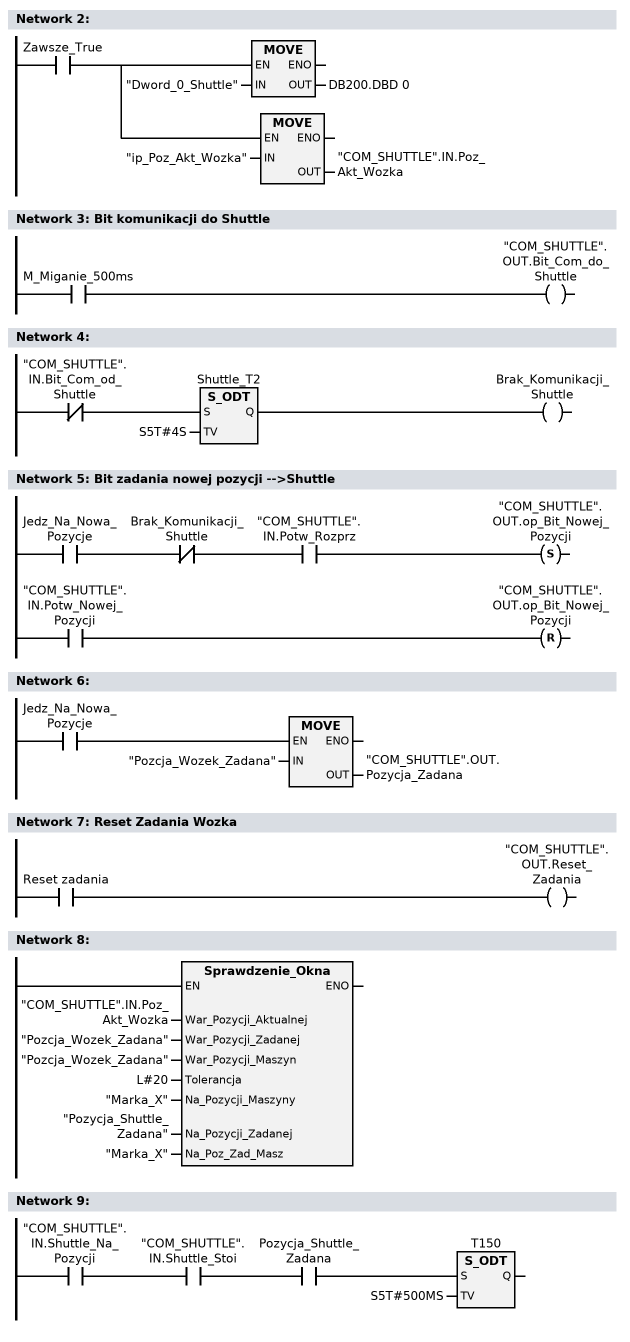
NETWORK
TITLE =
//przepisanie bitow wejsciowych s shuttle
      A     "Zawsze_True";
      =     L 0.0;
      A     L 0.0;
      JNB   _001;
      L     "Dword_0_Shuttle";
      T     DB200.DBD 0;
_001: NOP   0;
      A     L 0.0;
      JNB   _002;
      L     "ip_Poz_Akt_Wozka";
      T     "COM_SHUTTLE".IN.Poz_Akt_Wozka;
_002: NOP   0;
NETWORK
TITLE = Bit komunikacji do Shuttle
//Bit komunikacji z Shuttle          (i30.0 -q30.0)
//                                    (q38.0-i38.0)
      A     "M_Miganie_500ms";
      =     "COM_SHUTTLE".OUT.Bit_Com_do_Shuttle;
NETWORK
TITLE =
//Sprawdzenie komunikacji
      AN    "COM_SHUTTLE".IN.Bit_Com_od_Shuttle;
      L     S5T#4S;
      SD    "Shuttle_T2";
      NOP   0;
      NOP   0;
      NOP   0;
      A     "Shuttle_T2";
      =     "Brak_Komunikacji_Shuttle";
NETWORK
TITLE = Bit zadania nowej pozycji -->Shuttle
//Jazda na nowa pozycje             (q39.1 - i39.1)
//                                  (i31.1 - q31.1)
      A     "Jedz_Na_Nowa_Pozycje";
      AN    "Brak_Komunikacji_Shuttle";
      A     "COM_SHUTTLE".IN.Potw_Rozprz;
      S     "COM_SHUTTLE".OUT.op_Bit_Nowej_Pozycji;
      A     "COM_SHUTTLE".IN.Potw_Nowej_Pozycji;
      R     "COM_SHUTTLE".OUT.op_Bit_Nowej_Pozycji;
      NOP   0;
NETWORK
TITLE =
//Jedz na pozycje                  (qd42-id42)
      A     "Jedz_Na_Nowa_Pozycje";
      JNB   _003;
      L     "Pozcja_Wozek_Zadana";
      T     "COM_SHUTTLE".OUT.Pozycja_Zadana;
_003: NOP   0;
NETWORK
TITLE = Reset Zadania Wozka
      A     "Reset zadania";
      =     "COM_SHUTTLE".OUT.Reset_Zadania;
NETWORK
TITLE =
      CALL  "Sprawdzenie_Okna" (
           War_Pozycji_Aktualnej    := "COM_SHUTTLE".IN.Poz_Akt_Wozka,
           War_Pozycji_Zadanej      := "Pozcja_Wozek_Zadana",
           War_Pozycji_Maszyn       := "Pozcja_Wozek_Zadana",
           Tolerancja               := L#20,
           Na_Pozycji_Maszyny       := "Marka_X",
           Na_Pozycji_Zadanej       := "Pozycja_Shuttle_Zadana",
           Na_Poz_Zad_Masz          := "Marka_X");
      NOP   0;
NETWORK
TITLE =
//opoznienie potwierdzenia pozycji
      A     "COM_SHUTTLE".IN.Shuttle_Na_Pozycji;
      A     "COM_SHUTTLE".IN.Shuttle_Stoi;
      A     "Pozycja_Shuttle_Zadana";
      L     S5T#500MS;
      SD    "T150";
      NOP   0;
      NOP   0;
      NOP   0;
      NOP   0;
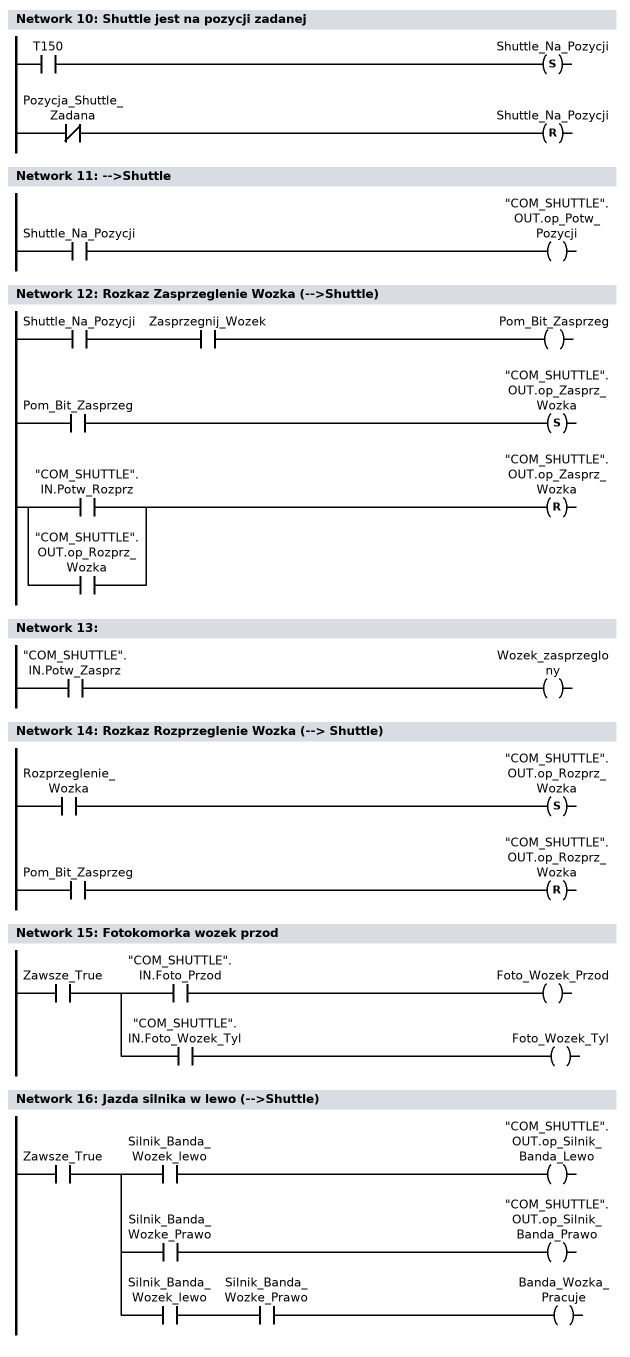
NETWORK
TITLE = Shuttle jest na pozycji zadanej
//Maszyna na pozcyji
      A     "T150";
      S     "Shuttle_Na_Pozycji";
      AN    "Pozycja_Shuttle_Zadana";
      R     "Shuttle_Na_Pozycji";
      NOP   0;
NETWORK
TITLE = -->Shuttle
//Potwierdzenie pozycji do shuttle
      A     "Shuttle_Na_Pozycji";
      =     "COM_SHUTTLE".OUT.op_Potw_Pozycji;
NETWORK
TITLE = Rozkaz Zasprzeglenie Wozka (-->Shuttle)
//Zasprzeglenie wozka Shuttle
      A     "Shuttle_Na_Pozycji";
      A     "Zasprzegnij_Wozek";
      =     "Pom_Bit_Zasprzeg";
      A     "Pom_Bit_Zasprzeg";
      S     "COM_SHUTTLE".OUT.op_Zasprz_Wozka;
      A(;
      O     "COM_SHUTTLE".IN.Potw_Rozprz;
      O     "COM_SHUTTLE".OUT.op_Rozprz_Wozka;
      );
      R     "COM_SHUTTLE".OUT.op_Zasprz_Wozka;
      NOP   0;
NETWORK
TITLE =
//Potwierdzenie zasprzeglenia wozka
      A     "COM_SHUTTLE".IN.Potw_Zasprz;
      =     "Wozek_zasprzeglony";
NETWORK
TITLE = Rozkaz Rozprzeglenie Wozka (--> Shuttle)
//Rozprzeglenie wozka
      A     "Rozprzeglenie_Wozka";
      S     "COM_SHUTTLE".OUT.op_Rozprz_Wozka;
      A     "Pom_Bit_Zasprzeg";
      R     "COM_SHUTTLE".OUT.op_Rozprz_Wozka;
      NOP   0;
NETWORK
TITLE = Fotokomorka wozek przod
//Przejecie fotokomorek
      A     "Zawsze_True";
      =     L 0.0;
      A     L 0.0;
      A     "COM_SHUTTLE".IN.Foto_Przod;
      =     "Foto_Wozek_Przod";
      A     L 0.0;
      A     "COM_SHUTTLE".IN.Foto_Wozek_Tyl;
      =     "Foto_Wozek_Tyl";
NETWORK
TITLE = Jazda silnika w lewo (-->Shuttle)
//Jazda silnikami
      A     "Zawsze_True";
      =     L 0.0;
      A     L 0.0;
      A     "Silnik_Banda_Wozek_lewo";
      =     "COM_SHUTTLE".OUT.op_Silnik_Banda_Lewo;
      A     L 0.0;
      A     "Silnik_Banda_Wozke_Prawo";
      =     "COM_SHUTTLE".OUT.op_Silnik_Banda_Prawo;
      A     L 0.0;
      A     "Silnik_Banda_Wozek_lewo";
      A     "Silnik_Banda_Wozke_Prawo";
      =     "Banda_Wozka_Pracuje";
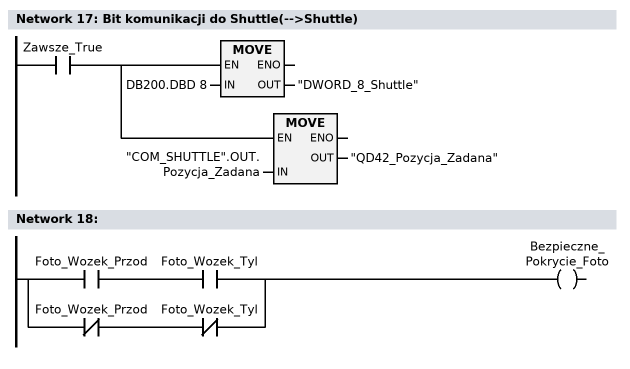
NETWORK
TITLE = Bit komunikacji do Shuttle(-->Shuttle)
//Przypisanie wyjsc
      A     "Zawsze_True";
      =     L 0.0;
      A     L 0.0;
      JNB   _004;
      L     DB200.DBD 8;
      T     "DWORD_8_Shuttle";
_004: NOP   0;
      A     L 0.0;
      JNB   _005;
      L     "COM_SHUTTLE".OUT.Pozycja_Zadana;
      T     "QD42_Pozycja_Zadana";
_005: NOP   0;
NETWORK
TITLE =
//foto bezpieczne
//
      A     "Foto_Wozek_Przod";
      A     "Foto_Wozek_Tyl";
      O;
      AN    "Foto_Wozek_Przod";
      AN    "Foto_Wozek_Tyl";
      =     "Bezpieczne_Pokrycie_Foto";
END_FUNCTION

FUNCTION "Wymiana_Pakietow_Wozek" : VOID	// FC 201
//Funkcja odpowiada za wymine duzej ilosci danych z wozkiem. Dane sa zapisywane 
//do 
//bloku LLIN. Wysylanie danych odbywa sie przy uzyciu bloku LLOUT. 
//
//Zmienne default- pobierane sa z kopii bloku z wartosciami stalymi i kopiowane 
//sa 
//do bloku roboczego (db800).Warunkiem poprawnego dzialania programu jest zasada 
//ze blok roboczy musi byc wiekszy od bloku pobieranego ,defaulotwego oraz 
//wysylanego. 
//
//Przycisk DEFAULT--> kopia np.db720 do db800(roboczy)
//Przycisk READ-->pobiera np.db720(shuttle) do db800(roboczy)
//Przycisk WRITE-->wysyla blok np.db800 do db720 shuttle.
//
//
//
VERSION : 0.1
BEGIN
NETWORK
TITLE =
//Ten network celowo jest wolny
//inputy to i160
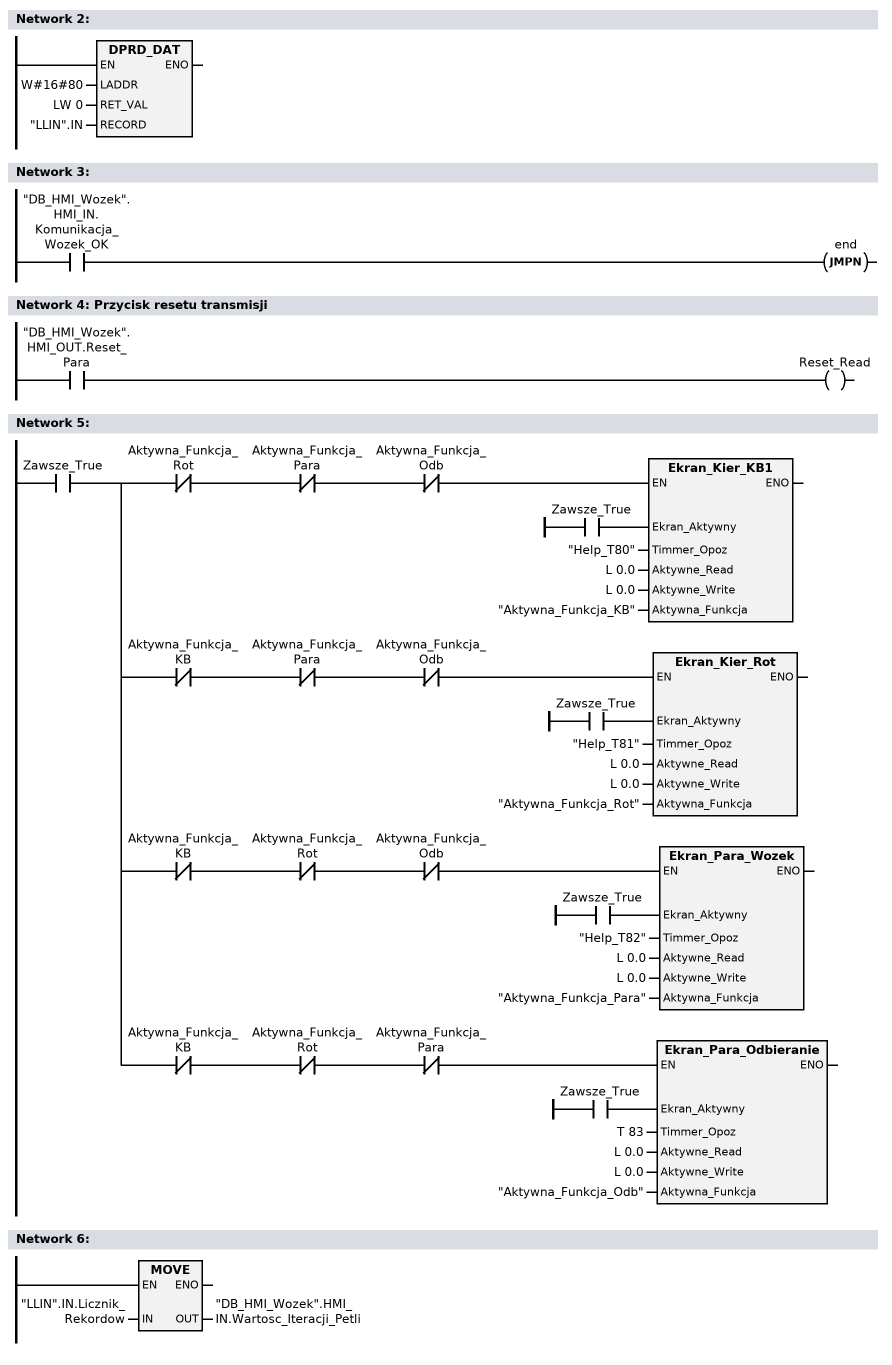
NETWORK
TITLE =
//Pobieranie danych
      CALL  "DPRD_DAT" (
           LADDR                    := W#16#80,
           RET_VAL                  := LW 0,
           RECORD                   := "LLIN".IN);
      NOP   0;
NETWORK
TITLE =
      A     "DB_HMI_Wozek".HMI_IN.Komunikacja_Wozek_OK;
      JCN   end;
NETWORK
TITLE = Przycisk resetu transmisji
//Resetowanie transmisji
      A     "DB_HMI_Wozek".HMI_OUT.Reset_Para;
      =     "Reset_Read";
NETWORK
TITLE =
      A     "Zawsze_True";
      =     L 2.0;
      A     "Zawsze_True";
      =     L 2.1;
      BLD   103;
      A     L 2.0;
      AN    "Aktywna_Funkcja_Rot";
      AN    "Aktywna_Funkcja_Para";
      AN    "Aktywna_Funkcja_Odb";
      JNB   _001;
      CALL  "Ekran_Kier_KB1" (
           Ekran_Aktywny            := L 2.1,
           Timmer_Opoz              := "Help_T80",
           Aktywne_Read             := L 0.0,
           Aktywne_Write            := L 0.0,
           Aktywna_Funkcja          := "Aktywna_Funkcja_KB");
_001: NOP   0;
      A     "Zawsze_True";
      =     L 2.1;
      BLD   103;
      A     L 2.0;
      AN    "Aktywna_Funkcja_KB";
      AN    "Aktywna_Funkcja_Para";
      AN    "Aktywna_Funkcja_Odb";
      JNB   _002;
      CALL  "Ekran_Kier_Rot" (
           Ekran_Aktywny            := L 2.1,
           Timmer_Opoz              := "Help_T81",
           Aktywne_Read             := L 0.0,
           Aktywne_Write            := L 0.0,
           Aktywna_Funkcja          := "Aktywna_Funkcja_Rot");
_002: NOP   0;
      A     "Zawsze_True";
      =     L 2.1;
      BLD   103;
      A     L 2.0;
      AN    "Aktywna_Funkcja_KB";
      AN    "Aktywna_Funkcja_Rot";
      AN    "Aktywna_Funkcja_Odb";
      JNB   _003;
      CALL  "Ekran_Para_Wozek" (
           Ekran_Aktywny            := L 2.1,
           Timmer_Opoz              := "Help_T82",
           Aktywne_Read             := L 0.0,
           Aktywne_Write            := L 0.0,
           Aktywna_Funkcja          := "Aktywna_Funkcja_Para");
_003: NOP   0;
      A     "Zawsze_True";
      =     L 2.1;
      BLD   103;
      A     L 2.0;
      AN    "Aktywna_Funkcja_KB";
      AN    "Aktywna_Funkcja_Rot";
      AN    "Aktywna_Funkcja_Para";
      JNB   _004;
      CALL  "Ekran_Para_Odbieranie" (
           Ekran_Aktywny            := L 2.1,
           Timmer_Opoz              := T 83,
           Aktywne_Read             := L 0.0,
           Aktywne_Write            := L 0.0,
           Aktywna_Funkcja          := "Aktywna_Funkcja_Odb");
_004: NOP   0;
NETWORK
TITLE =
      L     "LLIN".IN.Licznik_Rekordow;
      T     "DB_HMI_Wozek".HMI_IN.Wartosc_Iteracji_Petli;
      NOP   0;
NETWORK
TITLE =
end:  NOP   0;
// koniec
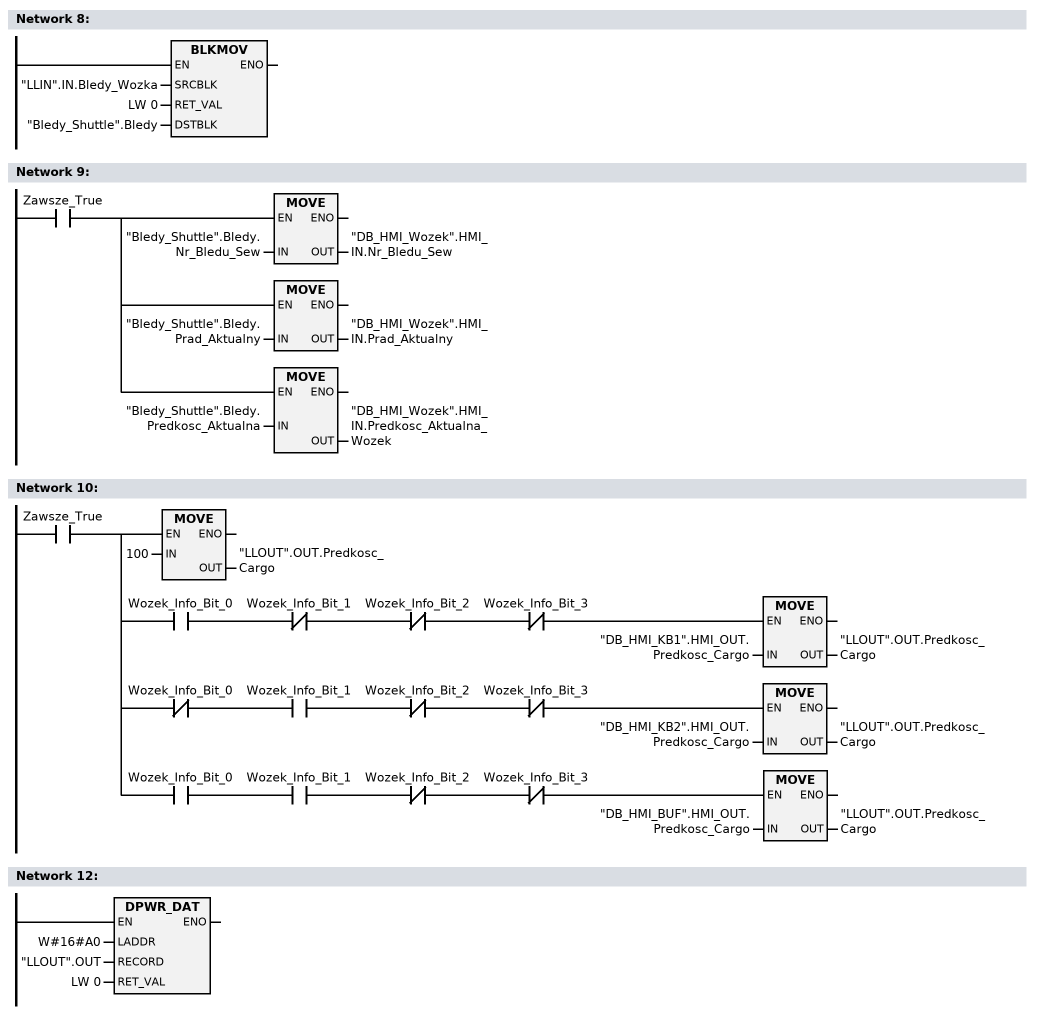
NETWORK
TITLE =
//Kopiowanie bledow wozka s
      CALL  "BLKMOV" (
           SRCBLK                   := "LLIN".IN.Bledy_Wozka,
           RET_VAL                  := LW 0,
           DSTBLK                   := "Bledy_Shuttle".Bledy);
      NOP   0;
NETWORK
TITLE =
//Niektore parametry wozka
      A     "Zawsze_True";
      =     L 2.0;
      A     L 2.0;
      JNB   _005;
      L     "Bledy_Shuttle".Bledy.Nr_Bledu_Sew;
      T     "DB_HMI_Wozek".HMI_IN.Nr_Bledu_Sew;
_005: NOP   0;
      A     L 2.0;
      JNB   _006;
      L     "Bledy_Shuttle".Bledy.Prad_Aktualny;
      T     "DB_HMI_Wozek".HMI_IN.Prad_Aktualny;
_006: NOP   0;
      A     L 2.0;
      JNB   _007;
      L     "Bledy_Shuttle".Bledy.Predkosc_Aktualna;
      T     "DB_HMI_Wozek".HMI_IN.Predkosc_Aktualna_Wozek;
_007: NOP   0;
NETWORK
TITLE =
//Wyslanie do wozka informacji o predkosci Cargo. W zaleznosci skad jest ladunek
      A     "Zawsze_True";
      =     L 2.0;
      A     L 2.0;
      JNB   _008;
      L     100;
      T     "LLOUT".OUT.Predkosc_Cargo;
_008: NOP   0;
      A     L 2.0;
      A     "Wozek_Info_Bit_0";
      AN    "Wozek_Info_Bit_1";
      AN    "Wozek_Info_Bit_2";
      AN    "Wozek_Info_Bit_3";
      JNB   _009;
      L     "DB_HMI_KB1".HMI_OUT.Predkosc_Cargo;
      T     "LLOUT".OUT.Predkosc_Cargo;
_009: NOP   0;
      A     L 2.0;
      AN    "Wozek_Info_Bit_0";
      A     "Wozek_Info_Bit_1";
      AN    "Wozek_Info_Bit_2";
      AN    "Wozek_Info_Bit_3";
      JNB   _00a;
      L     "DB_HMI_KB2".HMI_OUT.Predkosc_Cargo;
      T     "LLOUT".OUT.Predkosc_Cargo;
_00a: NOP   0;
      A     L 2.0;
      A     "Wozek_Info_Bit_0";
      A     "Wozek_Info_Bit_1";
      AN    "Wozek_Info_Bit_2";
      AN    "Wozek_Info_Bit_3";
      JNB   _00b;
      L     "DB_HMI_BUF".HMI_OUT.Predkosc_Cargo;
      T     "LLOUT".OUT.Predkosc_Cargo;
_00b: NOP   0;
NETWORK
TITLE =
NETWORK
TITLE =
//Wyslanie danych do wozka 
      CALL  "DPWR_DAT" (
           LADDR                    := W#16#A0,
           RECORD                   := "LLOUT".OUT,
           RET_VAL                  := LW 0);
      NOP   0;
END_FUNCTION

FUNCTION "Komunikacja_Gender" : VOID	// FC 205
//Marki 400. Bity sa widziane od strony odbierania
VERSION : 0.1
BEGIN
NETWORK
TITLE =
//Ten Network celowo jest wolny
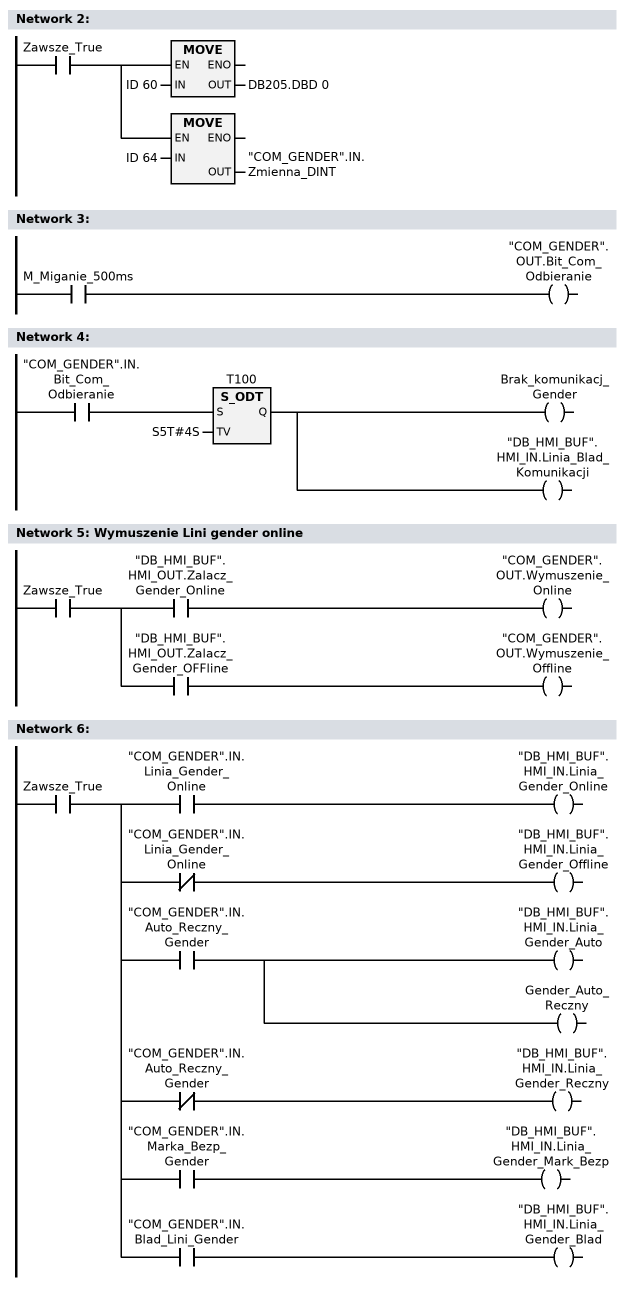
NETWORK
TITLE =
//Przypisanie danych z dp coupler
      A     "Zawsze_True";
      =     L 0.0;
      A     L 0.0;
      JNB   _001;
      L     ID 60;
      T     DB205.DBD 0;
_001: NOP   0;
      A     L 0.0;
      JNB   _002;
      L     ID 64;
      T     "COM_GENDER".IN.Zmienna_DINT;
_002: NOP   0;
NETWORK
TITLE =
//Komunikacj z Gender
      A     "M_Miganie_500ms";
      =     "COM_GENDER".OUT.Bit_Com_Odbieranie;
NETWORK
TITLE =
//Sprawdzenie czy komunikacja jest OK
      A     "COM_GENDER".IN.Bit_Com_Odbieranie;
      L     S5T#4S;
      SD    "T100";
      NOP   0;
      NOP   0;
      NOP   0;
      A     "T100";
      =     "Brak_komunikacj_Gender";
      =     "DB_HMI_BUF".HMI_IN.Linia_Blad_Komunikacji;
NETWORK
TITLE = Wymuszenie Lini gender online
//Wymus online/offline
      A     "Zawsze_True";
      =     L 0.0;
      A     L 0.0;
      A     "DB_HMI_BUF".HMI_OUT.Zalacz_Gender_Online;
      =     "COM_GENDER".OUT.Wymuszenie_Online;
      A     L 0.0;
      A     "DB_HMI_BUF".HMI_OUT.Zalacz_Gender_OFFline;
      =     "COM_GENDER".OUT.Wymuszenie_Offline;
NETWORK
TITLE =
//Wyswietlenie stanu pracy
      A     "Zawsze_True";
      =     L 0.0;
      A     L 0.0;
      A     "COM_GENDER".IN.Linia_Gender_Online;
      =     "DB_HMI_BUF".HMI_IN.Linia_Gender_Online;
      A     L 0.0;
      AN    "COM_GENDER".IN.Linia_Gender_Online;
      =     "DB_HMI_BUF".HMI_IN.Linia_Gender_Offline;
      A     L 0.0;
      A     "COM_GENDER".IN.Auto_Reczny_Gender;
      =     "DB_HMI_BUF".HMI_IN.Linia_Gender_Auto;
      =     "Gender_Auto_Reczny";
      A     L 0.0;
      AN    "COM_GENDER".IN.Auto_Reczny_Gender;
      =     "DB_HMI_BUF".HMI_IN.Linia_Gender_Reczny;
      A     L 0.0;
      A     "COM_GENDER".IN.Marka_Bezp_Gender;
      =     "DB_HMI_BUF".HMI_IN.Linia_Gender_Mark_Bezp;
      A     L 0.0;
      A     "COM_GENDER".IN.Blad_Lini_Gender;
      =     "DB_HMI_BUF".HMI_IN.Linia_Gender_Blad;
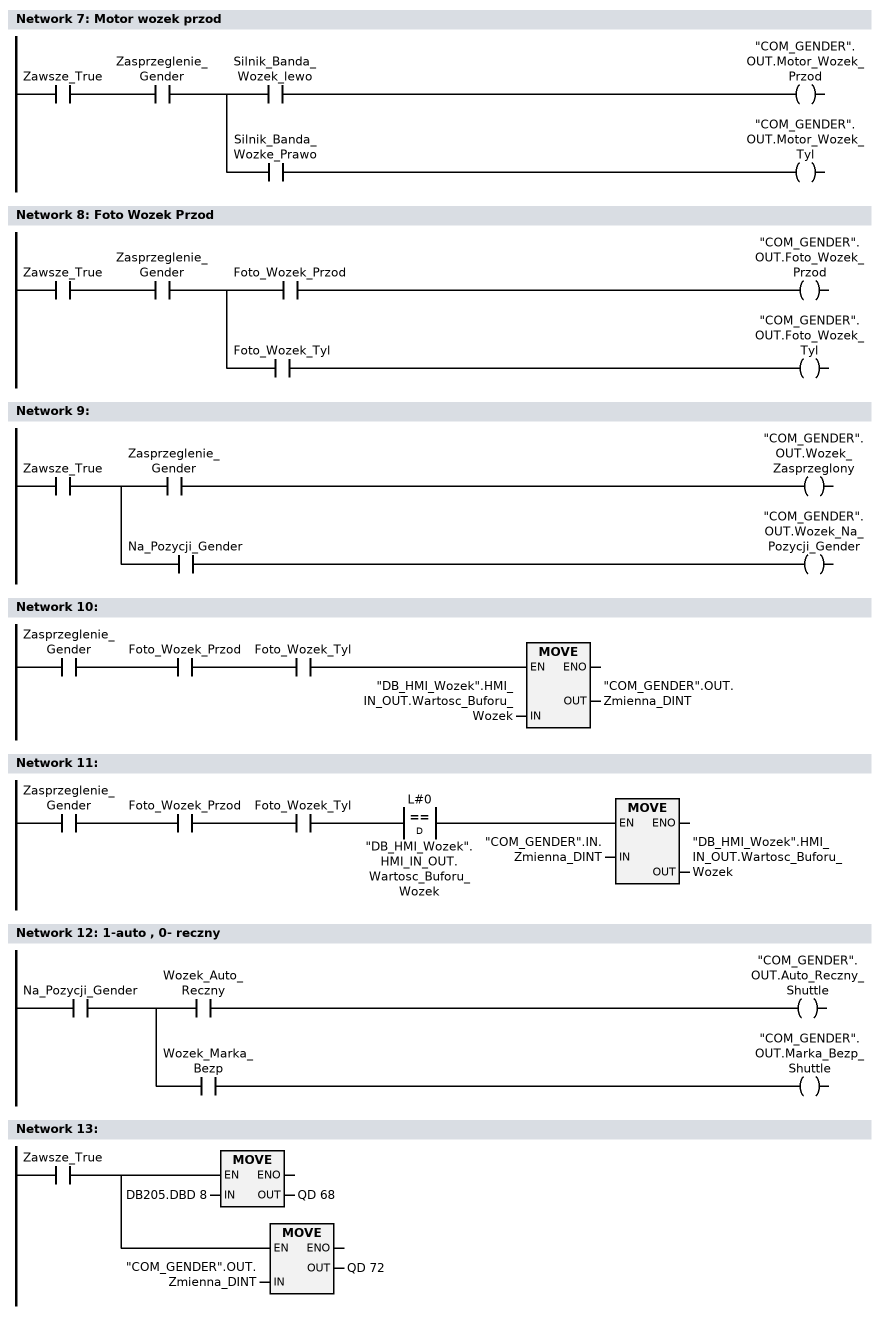
NETWORK
TITLE = Motor wozek przod
//Sygnaly silnika wozka 
      A     "Zawsze_True";
      A     "Zasprzeglenie_Gender";
      =     L 0.0;
      A     L 0.0;
      A     "Silnik_Banda_Wozek_lewo";
      =     "COM_GENDER".OUT.Motor_Wozek_Przod;
      A     L 0.0;
      A     "Silnik_Banda_Wozke_Prawo";
      =     "COM_GENDER".OUT.Motor_Wozek_Tyl;
NETWORK
TITLE = Foto Wozek Przod
      A     "Zawsze_True";
      A     "Zasprzeglenie_Gender";
      =     L 0.0;
      A     L 0.0;
      A     "Foto_Wozek_Przod";
      =     "COM_GENDER".OUT.Foto_Wozek_Przod;
      A     L 0.0;
      A     "Foto_Wozek_Tyl";
      =     "COM_GENDER".OUT.Foto_Wozek_Tyl;
NETWORK
TITLE =
//Sprawdzenie zasprzeglenia
      A     "Zawsze_True";
      =     L 0.0;
      A     L 0.0;
      A     "Zasprzeglenie_Gender";
      =     "COM_GENDER".OUT.Wozek_Zasprzeglony;
      A     L 0.0;
      A     "Na_Pozycji_Gender";
      =     "COM_GENDER".OUT.Wozek_Na_Pozycji_Gender;
NETWORK
TITLE =
      A     "Zasprzeglenie_Gender";
      A     "Foto_Wozek_Przod";
      A     "Foto_Wozek_Tyl";
      JNB   _003;
      L     "DB_HMI_Wozek".HMI_IN_OUT.Wartosc_Buforu_Wozek;
      T     "COM_GENDER".OUT.Zmienna_DINT;
_003: NOP   0;
NETWORK
TITLE =
//Gdy np jazda do tylu
      A     "Zasprzeglenie_Gender";
      A     "Foto_Wozek_Przod";
      A     "Foto_Wozek_Tyl";
      A(;
      L     L#0;
      L     "DB_HMI_Wozek".HMI_IN_OUT.Wartosc_Buforu_Wozek;
      ==D;
      );
      JNB   _004;
      L     "COM_GENDER".IN.Zmienna_DINT;
      T     "DB_HMI_Wozek".HMI_IN_OUT.Wartosc_Buforu_Wozek;
_004: NOP   0;
NETWORK
TITLE = 1-auto , 0- reczny
      A     "Na_Pozycji_Gender";
      =     L 0.0;
      A     L 0.0;
      A     "Wozek_Auto_Reczny";
      =     "COM_GENDER".OUT.Auto_Reczny_Shuttle;
      A     L 0.0;
      A     "Wozek_Marka_Bezp";
      =     "COM_GENDER".OUT.Marka_Bezp_Shuttle;
NETWORK
TITLE =
//Przypisanie danych z dp coupler
      A     "Zawsze_True";
      =     L 0.0;
      A     L 0.0;
      JNB   _005;
      L     DB205.DBD 8;
      T     QD 68;
_005: NOP   0;
      A     L 0.0;
      JNB   _006;
      L     "COM_GENDER".OUT.Zmienna_DINT;
      T     QD 72;
_006: NOP   0;
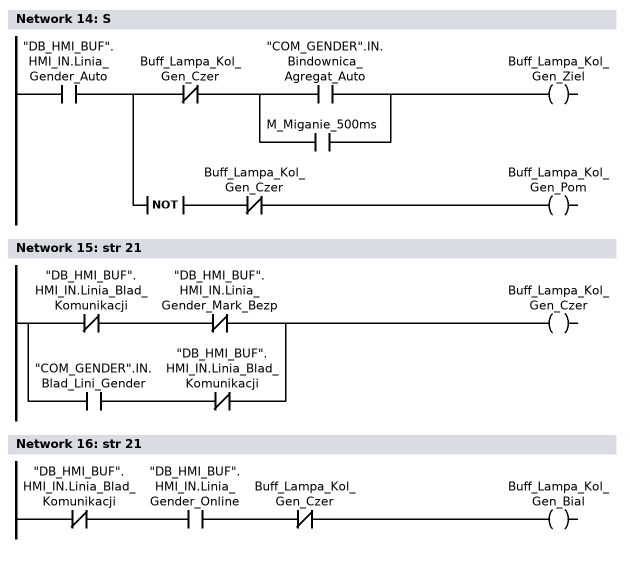
NETWORK
TITLE = S
//Dodanie lampek Gender
      A     "DB_HMI_BUF".HMI_IN.Linia_Gender_Auto;
      =     L 0.0;
      A     L 0.0;
      AN    "Buff_Lampa_Kol_Gen_Czer";
      A(;
      O     "COM_GENDER".IN.Bindownica_Agregat_Auto;
      O     "M_Miganie_500ms";
      );
      =     "Buff_Lampa_Kol_Gen_Ziel";
      A     L 0.0;
      NOT;
      AN    "Buff_Lampa_Kol_Gen_Czer";
      =     "Buff_Lampa_Kol_Gen_Pom";
NETWORK
TITLE = str 21
      AN    "DB_HMI_BUF".HMI_IN.Linia_Blad_Komunikacji;
      AN    "DB_HMI_BUF".HMI_IN.Linia_Gender_Mark_Bezp;
      O;
      A     "COM_GENDER".IN.Blad_Lini_Gender;
      AN    "DB_HMI_BUF".HMI_IN.Linia_Blad_Komunikacji;
      =     "Buff_Lampa_Kol_Gen_Czer";
NETWORK
TITLE = str 21
//Gender jest online
      AN    "DB_HMI_BUF".HMI_IN.Linia_Blad_Komunikacji;
      A     "DB_HMI_BUF".HMI_IN.Linia_Gender_Online;
      AN    "Buff_Lampa_Kol_Gen_Czer";
      =     "Buff_Lampa_Kol_Gen_Bial";
END_FUNCTION

FUNCTION "Monitor_Bandy" : VOID	// FC 313
//Funkcja na monitoruje przejezdzajacy miedzy bandami produkt
VERSION : 0.1
VAR_INPUT
  i_Foto_Koniec : BOOL ;
  i_Motor_Bandy : BOOL ;
  i_Zabierz_Od_Pop : BOOL ;	//Sygnal zabierz od bandy poprzedniej
  i_Zabierz_Do_Nast : BOOL ;	//Sygnal zabierz do nastepnej
  i_DW_Wartosc_Wej : DINT ;	//Wartosc wejsciowa z poprzedniej bandy
  i_Paleta_Dost_Od_Nast : BOOL ;
END_VAR
VAR_IN_OUT
  io_DW_Wartosc_Rej : DINT ;	//Wartosc bierzaca rejestru
  io_W_Pomoc : WORD ;	//Slowo pomocnicze
END_VAR
VAR_TEMP
  Rel_Z_Pop_Aktywna : BOOL ;	//Relacja z banda poprzednia jest aktywna
  Rel_Z_Nast_Aktywna : BOOL ;	//Relacja z banda nastepna jest aktywan
  Pom_LB1 : BYTE ;
  Pom_LW2 : WORD ;
  Pom_LD4 : BOOL ;
END_VAR
BEGIN
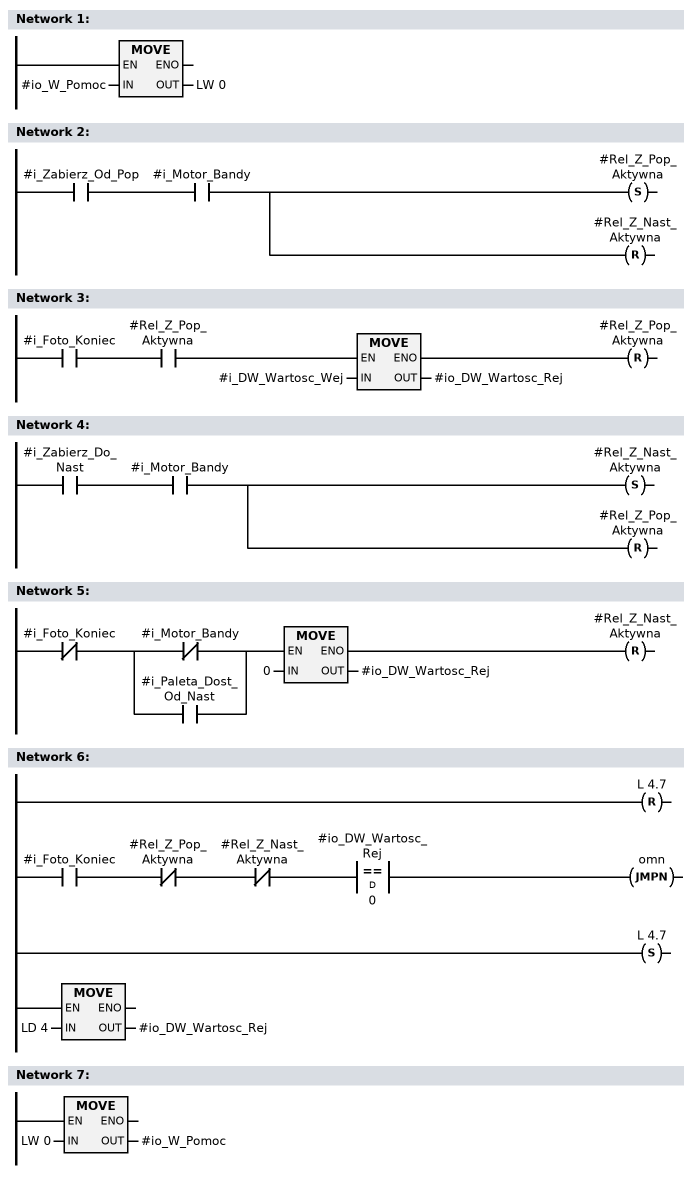
NETWORK
TITLE =
//Ten network celowo jest wolny
      L     #io_W_Pomoc;
      T     LW 0;
      NOP   0;
NETWORK
TITLE =
//Pobranie wartosci
      A     #i_Zabierz_Od_Pop;
      A     #i_Motor_Bandy;
      S     #Rel_Z_Pop_Aktywna;
      R     #Rel_Z_Nast_Aktywna;
NETWORK
TITLE =
//Dojazd do fotokomorki i przepisanie wartosci
      A     #i_Foto_Koniec;
      A     #Rel_Z_Pop_Aktywna;
      JNB   _001;
      L     #i_DW_Wartosc_Wej;
      T     #io_DW_Wartosc_Rej;
      SET;
      SAVE;
      CLR;
_001: A     BR;
      R     #Rel_Z_Pop_Aktywna;
NETWORK
TITLE =
//Relacja z nastepna banda
      A     #i_Zabierz_Do_Nast;
      A     #i_Motor_Bandy;
      S     #Rel_Z_Nast_Aktywna;
      R     #Rel_Z_Pop_Aktywna;
NETWORK
TITLE =
//Opuszczeni palety z bandy relacja przod
      AN    #i_Foto_Koniec;
      A(;
      ON    #i_Motor_Bandy;
      O     #i_Paleta_Dost_Od_Nast;
      );
      JNB   _002;
      L     0;
      T     #io_DW_Wartosc_Rej;
      SET;
      SAVE;
      CLR;
_002: A     BR;
      R     #Rel_Z_Nast_Aktywna;
NETWORK
TITLE =
//Nalozenie maski gdy jest paleta a wartosc rejsetru wskazuje na 0
//kasowanie bitu pomocniczego
      SET;
      R     L 4.7;
// Aby znalezc palete widmo
      A     #i_Foto_Koniec;
      AN    #Rel_Z_Pop_Aktywna;
      AN    #Rel_Z_Nast_Aktywna;
      A(;
      L     #io_DW_Wartosc_Rej;
      L     0;
      ==D;
      );
      JCN   omn;
      SET;
      S     L 4.7;	//najstarszy bit (info o palecie)
      L     LD 4;
      T     #io_DW_Wartosc_Rej;
omn:  NOP   0;
NETWORK
TITLE =
//Przypisanie wartosci z pamieci podrecznej
//
      L     LW 0;
      T     #io_W_Pomoc;
      NOP   0;
END_FUNCTION

FUNCTION "Monitor_Bandy_2" : VOID	// FC 314
//Funkcja na monitoruje przejezdzajacy miedzy bandami produkt
//Jezeli cos nie wyjdzie paleta widmo bierze wszystko na siebie
//
//
//0.7 - paleta obecna (nieuzywane)
//0.6 - kierunek spedycja (uzywane)
//0.5 - kierunek intro (uzywane)
//0.4 - wiazanie poprzeczne (uzywane)
//0.3 - wiazanie wzdluzne   (uzywane)
//0.2 - deklowanie (uzywane)
//0.1 - foliowanie (uzywane)
//0.0 - paleta obrabiana
//1.7 - rezerwa (nieuzywane)
//1.6 - rezerwa (nieuzywane)
//1.5 - rezerwa (nieuzywane)
//1.3 - rezerwa (nieuzywane)
//1.3 - info bit 3
//1.2 - info bit 2
//1.1 - info bit 1 
//1.0 - info bit 0
//
VERSION : 0.1
VAR_INPUT
  i_Auto_Reczny : BOOL ;	//1-Auto; 0-Reczny
  i_Foto_Tyl : BOOL ;
  i_Foto_Przod : BOOL ;
  i_Zabierz_Od_Pop : BOOL ;	//Sygnal zabierz od bandy poprzedniej
  i_Zabierz_Do_Nast : BOOL ;	//Sygnal zabierz do nastepnej
  i_Paleta_Dost_Od_Nast : BOOL ;
  i_Motor_Bandy_Przod : BOOL ;
  i_DW_Wartosc_Wej_Tyl : DINT ;	//Wartosc wejsciowa z poprzedniej bandy
  i_DW_Wartosc_Wej_Przod : DINT ;
  Timmer_Kontroli : TIMER ;
END_VAR
VAR_IN_OUT
  io_DW_Wartosc_Rej : DINT ;	//Wartosc bierzaca rejestru
  io_W_Pomoc : WORD ;	//Slowo pomocnicze
END_VAR
VAR_TEMP
  Rel_Z_Pop_Aktywna : BOOL ;	//Relacja z banda poprzednia jest aktywna
  Rel_Z_Nast_Aktywna : BOOL ;	//Relacja z banda nastepna jest aktywan
  Help_Zbocze_1 : BOOL ;
  Help_Zbocze_2 : BOOL ;
  Help_Zbocze_3 : BOOL ;
  Help_Zbocze_4 : BOOL ;
  Help_Zbocze_5 : BOOL ;
  Pom_LB1 : BYTE ;
  Pom_LW2 : WORD ;
  Pom_LD4 : DINT ;
  Pom_LD8 : DINT ;
END_VAR
BEGIN
